(* IEC 61131-3 sources: SmartHomeNew/ (part 6) *)

(* ---- FB_Heating_Runtime_Explainability_Publisher.st ---- *)
FUNCTION_BLOCK FB_Heating_Runtime_Explainability_Publisher
VAR_INPUT
    VI_Enable : BOOL;
    VI_System_Time_MS : UDINT;
    VI_Runtime_Context : ST_Heating_Runtime_Context;
    VI_Runtime_Observation_Valid : BOOL;
    VI_Runtime_Observer_Fault : BOOL;
    VI_Runtime_Status_Code : UINT;
    VI_Runtime_Status_Text : STRING(128);
END_VAR
VAR_OUTPUT
    VO_Phase_Event : ST_Heating_Runtime_Phase_Event;
    VO_Anomaly : ST_Heating_Runtime_Anomaly;
    VO_Blackbox_Event : ST_Heating_Runtime_Blackbox_Event;
    VO_Blackbox_Timeline : ST_Heating_Runtime_Blackbox_Timeline;
    VO_Event_Buffer : ST_Heating_Runtime_Event_Buffer;
    VO_Adaptive_Intelligence : ST_Heating_Runtime_Adaptive_Intelligence;
    VO_Causality_Graph : ST_Heating_Runtime_Causality_Graph;
    VO_Integration_Bridge : ST_Heating_Runtime_Integration_Bridge;
    VO_Predictive_State : ST_Heating_Runtime_Predictive_State;
    VO_Execution_Timeline : ST_Heating_Runtime_Execution_Timeline;
    VO_Phase_Transition : ST_Heating_Runtime_Phase_Transition;
    VO_Publication_Valid : BOOL;
END_VAR
VAR
    L_Sequencing_Valid : BOOL;
    L_Ownership_Valid : BOOL;
    L_Synchronization_Valid : BOOL;
    L_Runtime_Degraded : BOOL;
    L_Status_Code : UINT;

    L_Empty_Phase_Event : ST_Heating_Runtime_Phase_Event;
    L_Empty_Anomaly : ST_Heating_Runtime_Anomaly;
    L_Empty_Blackbox_Event : ST_Heating_Runtime_Blackbox_Event;
    L_Empty_Blackbox_Timeline : ST_Heating_Runtime_Blackbox_Timeline;
    L_Empty_Event_Buffer : ST_Heating_Runtime_Event_Buffer;
    L_Empty_Adaptive_Intelligence : ST_Heating_Runtime_Adaptive_Intelligence;
    L_Empty_Causality_Graph : ST_Heating_Runtime_Causality_Graph;
    L_Empty_Integration_Bridge : ST_Heating_Runtime_Integration_Bridge;
    L_Empty_Predictive_State : ST_Heating_Runtime_Predictive_State;
    L_Empty_Execution_Timeline : ST_Heating_Runtime_Execution_Timeline;
    L_Empty_Phase_Transition : ST_Heating_Runtime_Phase_Transition;
END_VAR

// Clear complete retained output snapshots before writing current frame.
// This prevents stale array entries in timeline/event/causality structures.
VO_Phase_Event := L_Empty_Phase_Event;
VO_Anomaly := L_Empty_Anomaly;
VO_Blackbox_Event := L_Empty_Blackbox_Event;
VO_Blackbox_Timeline := L_Empty_Blackbox_Timeline;
VO_Event_Buffer := L_Empty_Event_Buffer;
VO_Adaptive_Intelligence := L_Empty_Adaptive_Intelligence;
VO_Causality_Graph := L_Empty_Causality_Graph;
VO_Integration_Bridge := L_Empty_Integration_Bridge;
VO_Predictive_State := L_Empty_Predictive_State;
VO_Execution_Timeline := L_Empty_Execution_Timeline;
VO_Phase_Transition := L_Empty_Phase_Transition;
VO_Publication_Valid := FALSE;

IF NOT VI_Enable THEN
    RETURN;
END_IF;

L_Sequencing_Valid := VI_Runtime_Context.DHW_Before_Heating_Valid AND VI_Runtime_Context.State_Publication_Before_Diagnostics_Valid;
L_Ownership_Valid := VI_Runtime_Context.OpenTherm_Ownership_Valid AND VI_Runtime_Context.Cascade_Ownership_Valid AND VI_Runtime_Context.Safety_Isolation_Valid;
L_Synchronization_Valid := VI_Runtime_Context.Output_Projection_Last_Valid;
L_Runtime_Degraded := VI_Runtime_Observer_Fault OR NOT VI_Runtime_Observation_Valid;
L_Status_Code := VI_Runtime_Status_Code;

// Phase event
VO_Phase_Event.Phase := VI_Runtime_Context.Current_Phase;
VO_Phase_Event.Event_Active := TRUE;
VO_Phase_Event.Event_Completed := VI_Runtime_Observation_Valid;
VO_Phase_Event.Event_Failed := VI_Runtime_Observer_Fault;
VO_Phase_Event.Start_Time_MS := VI_System_Time_MS;
VO_Phase_Event.End_Time_MS := VI_System_Time_MS;
VO_Phase_Event.Duration_MS := 0;
VO_Phase_Event.Ordering_Valid := VI_Runtime_Context.DHW_Before_Heating_Valid;
VO_Phase_Event.Isolation_Valid := VI_Runtime_Context.Diagnostics_Isolation_Valid;
VO_Phase_Event.Status_Code := L_Status_Code;
VO_Phase_Event.Status_Text := VI_Runtime_Status_Text;
VO_Phase_Event.Diagnostics_Visible := TRUE;
VO_Phase_Event.Explainability_Visible := TRUE;
VO_Phase_Event.Safety_Integrity_Valid := VI_Runtime_Context.Safety_Isolation_Valid;
VO_Phase_Event.OpenTherm_Ownership_Valid := VI_Runtime_Context.OpenTherm_Ownership_Valid;
VO_Phase_Event.Cascade_Ownership_Valid := VI_Runtime_Context.Cascade_Ownership_Valid;

// Phase transition snapshot
VO_Phase_Transition.Previous_Phase := VI_Runtime_Context.Current_Phase;
VO_Phase_Transition.Current_Phase := VI_Runtime_Context.Current_Phase;
VO_Phase_Transition.Next_Phase := VI_Runtime_Context.Current_Phase;
VO_Phase_Transition.Transition_Active := TRUE;
VO_Phase_Transition.Transition_Completed := VI_Runtime_Observation_Valid;
VO_Phase_Transition.Transition_Failed := VI_Runtime_Observer_Fault;
VO_Phase_Transition.Transition_Start_MS := VI_System_Time_MS;
VO_Phase_Transition.Transition_End_MS := VI_System_Time_MS;
VO_Phase_Transition.Transition_Duration_MS := 0;
VO_Phase_Transition.Sequencing_Valid := L_Sequencing_Valid;
VO_Phase_Transition.Ownership_Valid := L_Ownership_Valid;
VO_Phase_Transition.Synchronization_Valid := L_Synchronization_Valid;
VO_Phase_Transition.Status_Code := L_Status_Code;
VO_Phase_Transition.Status_Text := VI_Runtime_Status_Text;

// Anomaly
VO_Anomaly.Anomaly_Active := VI_Runtime_Observer_Fault;
VO_Anomaly.Anomaly_Acknowledged := FALSE;
VO_Anomaly.Anomaly_Cleared := NOT VI_Runtime_Observer_Fault;
VO_Anomaly.Runtime_Jitter_Detected := FALSE;
VO_Anomaly.Runtime_Latency_Detected := FALSE;
VO_Anomaly.Runtime_Degraded := L_Runtime_Degraded;
VO_Anomaly.Cascade_Degraded := NOT VI_Runtime_Context.Cascade_Ownership_Valid;
VO_Anomaly.Cascade_Boiler_Loss_Detected := FALSE;
VO_Anomaly.OpenTherm_Transport_Degraded := NOT VI_Runtime_Context.OpenTherm_Ownership_Valid;
VO_Anomaly.OpenTherm_Command_Invalid := FALSE;
VO_Anomaly.Diagnostics_Degraded := NOT VI_Runtime_Context.Diagnostics_Isolation_Valid;
VO_Anomaly.Explainability_Degraded := NOT VI_Runtime_Context.Explainability_Isolation_Valid;
VO_Anomaly.Sequencing_Invalid := NOT L_Sequencing_Valid;
VO_Anomaly.Ownership_Invalid := NOT L_Ownership_Valid;
VO_Anomaly.Synchronization_Invalid := NOT L_Synchronization_Valid;
VO_Anomaly.Severity_Level := SEL(VI_Runtime_Observer_Fault, 1, 900);
VO_Anomaly.Critical_Anomaly := VI_Runtime_Observer_Fault;
VO_Anomaly.Status_Code := L_Status_Code;
VO_Anomaly.Status_Text := VI_Runtime_Status_Text;

// Blackbox event
VO_Blackbox_Event.Event_ID := VI_System_Time_MS;
VO_Blackbox_Event.Event_Active := TRUE;
VO_Blackbox_Event.Runtime_Phase := VI_Runtime_Context.Current_Phase;
VO_Blackbox_Event.Event_Start_MS := VI_System_Time_MS;
VO_Blackbox_Event.Event_End_MS := VI_System_Time_MS;
VO_Blackbox_Event.Event_Duration_MS := 0;
VO_Blackbox_Event.Runtime_Degraded := L_Runtime_Degraded;
VO_Blackbox_Event.Runtime_Fault := VI_Runtime_Observer_Fault;
VO_Blackbox_Event.Cascade_Degraded := NOT VI_Runtime_Context.Cascade_Ownership_Valid;
VO_Blackbox_Event.Cascade_Boiler_Loss := FALSE;
VO_Blackbox_Event.OpenTherm_Degraded := NOT VI_Runtime_Context.OpenTherm_Ownership_Valid;
VO_Blackbox_Event.OpenTherm_Command_Invalid := FALSE;
VO_Blackbox_Event.Sequencing_Invalid := NOT L_Sequencing_Valid;
VO_Blackbox_Event.Ownership_Invalid := NOT L_Ownership_Valid;
VO_Blackbox_Event.Synchronization_Invalid := NOT L_Synchronization_Valid;
VO_Blackbox_Event.Root_Cause_Candidate := VI_Runtime_Observer_Fault;
VO_Blackbox_Event.Critical_Path := VI_Runtime_Observer_Fault;
VO_Blackbox_Event.Status_Code := L_Status_Code;
VO_Blackbox_Event.Status_Text := VI_Runtime_Status_Text;

// Blackbox timeline snapshot
VO_Blackbox_Timeline.Write_Index := 1;
VO_Blackbox_Timeline.Event_Count := 1;
VO_Blackbox_Timeline.Timeline_Overflow := FALSE;
VO_Blackbox_Timeline.Reconstruction_Visible := TRUE;
VO_Blackbox_Timeline.Forensic_Timeline_Visible := TRUE;
VO_Blackbox_Timeline.Root_Cause_Reconstructed := VI_Runtime_Observer_Fault;
VO_Blackbox_Timeline.Sequencing_Valid := L_Sequencing_Valid;
VO_Blackbox_Timeline.Ownership_Valid := L_Ownership_Valid;
VO_Blackbox_Timeline.Synchronization_Valid := L_Synchronization_Valid;
VO_Blackbox_Timeline.Events[1] := VO_Blackbox_Event;
VO_Blackbox_Timeline.Status_Code := L_Status_Code;
VO_Blackbox_Timeline.Status_Text := VI_Runtime_Status_Text;

// Runtime event buffer snapshot
VO_Event_Buffer.Write_Index := 1;
VO_Event_Buffer.Read_Index := 1;
VO_Event_Buffer.Event_Count := 1;
VO_Event_Buffer.Overflow := FALSE;
VO_Event_Buffer.Ordering_Integrity_Valid := L_Sequencing_Valid;
VO_Event_Buffer.Isolation_Integrity_Valid := VI_Runtime_Context.Diagnostics_Isolation_Valid;
VO_Event_Buffer.Lifecycle_Integrity_Valid := VI_Runtime_Observation_Valid;
VO_Event_Buffer.Diagnostics_Visibility_Valid := TRUE;
VO_Event_Buffer.Explainability_Visibility_Valid := TRUE;
VO_Event_Buffer.OpenTherm_Ownership_Valid := VI_Runtime_Context.OpenTherm_Ownership_Valid;
VO_Event_Buffer.Cascade_Ownership_Valid := VI_Runtime_Context.Cascade_Ownership_Valid;
VO_Event_Buffer.Safety_Ownership_Valid := VI_Runtime_Context.Safety_Isolation_Valid;
VO_Event_Buffer.Events[1] := VO_Phase_Event;
VO_Event_Buffer.Status_Code := L_Status_Code;
VO_Event_Buffer.Status_Text := VI_Runtime_Status_Text;

// Passive integration bridge
VO_Integration_Bridge.Shell_Ready := VI_Runtime_Observation_Valid;
VO_Integration_Bridge.Shell_Fault := VI_Runtime_Observer_Fault;
VO_Integration_Bridge.Shell_Contract_Valid := VI_Runtime_Observation_Valid;
VO_Integration_Bridge.Allow_DHW_Integration := VI_Runtime_Context.Allow_DHW_Phase;
VO_Integration_Bridge.Allow_Heating_Integration := VI_Runtime_Context.Allow_Heating_Phase;
VO_Integration_Bridge.Allow_Diagnostics_Integration := VI_Runtime_Context.Allow_Diagnostics_Phase;
VO_Integration_Bridge.Allow_Output_Projection_Integration := VI_Runtime_Context.Allow_Output_Projection_Phase;
VO_Integration_Bridge.Runtime_Ownership_Valid := TRUE;
VO_Integration_Bridge.Diagnostics_Ownership_Valid := VI_Runtime_Context.Diagnostics_Isolation_Valid;
VO_Integration_Bridge.Explainability_Ownership_Valid := VI_Runtime_Context.Explainability_Isolation_Valid;
VO_Integration_Bridge.OpenTherm_Ownership_Valid := VI_Runtime_Context.OpenTherm_Ownership_Valid;
VO_Integration_Bridge.Cascade_Ownership_Valid := VI_Runtime_Context.Cascade_Ownership_Valid;
VO_Integration_Bridge.Safety_Ownership_Valid := VI_Runtime_Context.Safety_Isolation_Valid;
VO_Integration_Bridge.DHW_Before_Heating_Valid := VI_Runtime_Context.DHW_Before_Heating_Valid;
VO_Integration_Bridge.Diagnostics_After_Publication_Valid := VI_Runtime_Context.State_Publication_Before_Diagnostics_Valid;
VO_Integration_Bridge.Output_Projection_Last_Valid := VI_Runtime_Context.Output_Projection_Last_Valid;
VO_Integration_Bridge.Governance_Locked := TRUE;
VO_Integration_Bridge.Runtime_Attachment_Allowed := FALSE;
VO_Integration_Bridge.Runtime_Attachment_Active := FALSE;
VO_Integration_Bridge.Integration_Status_Code := L_Status_Code;
VO_Integration_Bridge.Integration_Status_Text := VI_Runtime_Status_Text;
VO_Integration_Bridge.Diagnostics_Visible := TRUE;
VO_Integration_Bridge.Explainability_Visible := TRUE;
VO_Integration_Bridge.Current_Phase := VI_Runtime_Context.Current_Phase;
VO_Integration_Bridge.Runtime_Synchronized := L_Synchronization_Valid;

// Predictive state (passive only)
VO_Predictive_State.Predictive_Analytics_Visible := TRUE;
VO_Predictive_State.Predictive_Analytics_Degraded := L_Runtime_Degraded;
VO_Predictive_State.Predictive_Analytics_Attention := NOT VI_Runtime_Observation_Valid;
VO_Predictive_State.Runtime_Stable := NOT L_Runtime_Degraded;
VO_Predictive_State.Runtime_Stability_Score := SEL(L_Runtime_Degraded, 100, 900);
VO_Predictive_State.Runtime_Degradation_Observation := SEL(L_Runtime_Degraded, 0, 900);
VO_Predictive_State.Runtime_Failure_Observation := SEL(VI_Runtime_Observer_Fault, 0, 900);
VO_Predictive_State.Cascade_Degradation_Observation := SEL(VI_Runtime_Context.Cascade_Ownership_Valid, 900, 0);
VO_Predictive_State.Cascade_Degraded_Trend_Visible := TRUE;
VO_Predictive_State.OpenTherm_Instability_Observation := SEL(VI_Runtime_Context.OpenTherm_Ownership_Valid, 900, 0);
VO_Predictive_State.OpenTherm_Degraded_Trend_Visible := TRUE;
VO_Predictive_State.Sequencing_Observation := SEL(L_Sequencing_Valid, 900, 0);
VO_Predictive_State.Ownership_Observation := SEL(L_Ownership_Valid, 900, 0);
VO_Predictive_State.Synchronization_Observation := SEL(L_Synchronization_Valid, 900, 0);
VO_Predictive_State.Status_Code := L_Status_Code;
VO_Predictive_State.Status_Text := VI_Runtime_Status_Text;

// Execution timeline snapshot
VO_Execution_Timeline.Write_Index := 1;
VO_Execution_Timeline.Frame_Count := 1;
VO_Execution_Timeline.Timeline_Overflow := FALSE;
VO_Execution_Timeline.Sequencing_Valid := L_Sequencing_Valid;
VO_Execution_Timeline.Ownership_Valid := L_Ownership_Valid;
VO_Execution_Timeline.Synchronization_Valid := L_Synchronization_Valid;
VO_Execution_Timeline.Runtime_Jitter_Detected := FALSE;
VO_Execution_Timeline.Runtime_Latency_Detected := FALSE;
VO_Execution_Timeline.Runtime_Degraded := L_Runtime_Degraded;
VO_Execution_Timeline.Frames[1].Phase := VI_Runtime_Context.Current_Phase;
VO_Execution_Timeline.Frames[1].Frame_Started := TRUE;
VO_Execution_Timeline.Frames[1].Frame_Completed := VI_Runtime_Observation_Valid;
VO_Execution_Timeline.Frames[1].Frame_Failed := VI_Runtime_Observer_Fault;
VO_Execution_Timeline.Frames[1].Frame_Start_MS := VI_System_Time_MS;
VO_Execution_Timeline.Frames[1].Frame_End_MS := VI_System_Time_MS;
VO_Execution_Timeline.Frames[1].Frame_Duration_MS := 0;
VO_Execution_Timeline.Frames[1].Sequencing_Valid := L_Sequencing_Valid;
VO_Execution_Timeline.Frames[1].Ownership_Valid := L_Ownership_Valid;
VO_Execution_Timeline.Frames[1].Synchronization_Valid := L_Synchronization_Valid;
VO_Execution_Timeline.Frames[1].Runtime_Jitter_Detected := FALSE;
VO_Execution_Timeline.Frames[1].Runtime_Latency_Detected := FALSE;
VO_Execution_Timeline.Frames[1].Runtime_Degraded := L_Runtime_Degraded;
VO_Execution_Timeline.Frames[1].Status_Code := L_Status_Code;
VO_Execution_Timeline.Frames[1].Status_Text := VI_Runtime_Status_Text;
VO_Execution_Timeline.Status_Code := L_Status_Code;
VO_Execution_Timeline.Status_Text := VI_Runtime_Status_Text;

// Adaptive intelligence (passive only)
VO_Adaptive_Intelligence.Adaptive_Analytics_Visible := TRUE;
VO_Adaptive_Intelligence.Adaptive_Analytics_Degraded := L_Runtime_Degraded;
VO_Adaptive_Intelligence.Adaptive_Analytics_Attention := NOT VI_Runtime_Observation_Valid;
VO_Adaptive_Intelligence.Supervision_Confidence_Observation := SEL(L_Runtime_Degraded, 100, 900);
VO_Adaptive_Intelligence.Confidence_Degradation_Visible := L_Runtime_Degraded;
VO_Adaptive_Intelligence.Adaptive_Runtime_Observation := 1;
VO_Adaptive_Intelligence.Adaptive_Runtime_Stability_Observation := SEL(L_Runtime_Degraded, 100, 900);
VO_Adaptive_Intelligence.Runtime_Anomaly_Observation_Weight := 1;
VO_Adaptive_Intelligence.Cascade_Anomaly_Observation_Weight := 1;
VO_Adaptive_Intelligence.OpenTherm_Anomaly_Observation_Weight := 1;
VO_Adaptive_Intelligence.Diagnostics_Anomaly_Observation_Weight := 1;
VO_Adaptive_Intelligence.Predictive_Correlation_Observation := 1;
VO_Adaptive_Intelligence.Predictive_Correlation_Visible := TRUE;
VO_Adaptive_Intelligence.Sequencing_Confidence_Observation := SEL(L_Sequencing_Valid, 100, 900);
VO_Adaptive_Intelligence.Ownership_Confidence_Observation := SEL(L_Ownership_Valid, 100, 900);
VO_Adaptive_Intelligence.Synchronization_Confidence_Observation := SEL(L_Synchronization_Valid, 100, 900);
VO_Adaptive_Intelligence.Status_Code := L_Status_Code;
VO_Adaptive_Intelligence.Status_Text := VI_Runtime_Status_Text;

// Minimal causality graph snapshot
VO_Causality_Graph.Node_Count := 1;
VO_Causality_Graph.Edge_Count := 1;
VO_Causality_Graph.Graph_Active := TRUE;
VO_Causality_Graph.Graph_Degraded := L_Runtime_Degraded;
VO_Causality_Graph.Graph_Critical := VI_Runtime_Observer_Fault;
VO_Causality_Graph.Sequencing_Valid := L_Sequencing_Valid;
VO_Causality_Graph.Ownership_Valid := L_Ownership_Valid;
VO_Causality_Graph.Synchronization_Valid := L_Synchronization_Valid;
VO_Causality_Graph.Nodes[1].Node_ID := 1;
VO_Causality_Graph.Nodes[1].Node_Active := TRUE;
VO_Causality_Graph.Nodes[1].Runtime_Degraded := L_Runtime_Degraded;
VO_Causality_Graph.Nodes[1].Runtime_Fault := VI_Runtime_Observer_Fault;
VO_Causality_Graph.Nodes[1].Cascade_Degraded := NOT VI_Runtime_Context.Cascade_Ownership_Valid;
VO_Causality_Graph.Nodes[1].OpenTherm_Degraded := NOT VI_Runtime_Context.OpenTherm_Ownership_Valid;
VO_Causality_Graph.Nodes[1].Diagnostics_Degraded := NOT VI_Runtime_Context.Diagnostics_Isolation_Valid;
VO_Causality_Graph.Nodes[1].Explainability_Degraded := NOT VI_Runtime_Context.Explainability_Isolation_Valid;
VO_Causality_Graph.Nodes[1].Sequencing_Invalid := NOT L_Sequencing_Valid;
VO_Causality_Graph.Nodes[1].Ownership_Invalid := NOT L_Ownership_Valid;
VO_Causality_Graph.Nodes[1].Synchronization_Invalid := NOT L_Synchronization_Valid;
VO_Causality_Graph.Nodes[1].Severity_Level := SEL(VI_Runtime_Observer_Fault, 1, 900);
VO_Causality_Graph.Nodes[1].Root_Cause_Candidate := VI_Runtime_Observer_Fault;
VO_Causality_Graph.Nodes[1].Status_Code := L_Status_Code;
VO_Causality_Graph.Nodes[1].Status_Text := VI_Runtime_Status_Text;
VO_Causality_Graph.Edges[1].Source_Node_ID := 1;
VO_Causality_Graph.Edges[1].Target_Node_ID := 1;
VO_Causality_Graph.Edges[1].Edge_Active := TRUE;
VO_Causality_Graph.Edges[1].Propagation_Detected := L_Runtime_Degraded;
VO_Causality_Graph.Edges[1].Runtime_Propagation := L_Runtime_Degraded;
VO_Causality_Graph.Edges[1].Cascade_Propagation := NOT VI_Runtime_Context.Cascade_Ownership_Valid;
VO_Causality_Graph.Edges[1].OpenTherm_Propagation := NOT VI_Runtime_Context.OpenTherm_Ownership_Valid;
VO_Causality_Graph.Edges[1].Diagnostics_Propagation := NOT VI_Runtime_Context.Diagnostics_Isolation_Valid;
VO_Causality_Graph.Edges[1].Sequencing_Propagation := NOT L_Sequencing_Valid;
VO_Causality_Graph.Edges[1].Ownership_Propagation := NOT L_Ownership_Valid;
VO_Causality_Graph.Edges[1].Synchronization_Propagation := NOT L_Synchronization_Valid;
VO_Causality_Graph.Status_Code := L_Status_Code;
VO_Causality_Graph.Status_Text := VI_Runtime_Status_Text;

VO_Publication_Valid := TRUE;

END_FUNCTION_BLOCK
// >>> BULK_SYNC_ANCHOR: FB_Heating_Runtime_Explainability_Publisher <<<

(* ---- FB_Heating_Runtime_Fault_Replay_Analyzer.st ---- *)
// ==============================================================================
// Heating runtime fault replay analyzer
// Read-only runtime forensic replay layer.
// ==============================================================================
FUNCTION_BLOCK FB_Heating_Runtime_Fault_Replay_Analyzer
VAR_INPUT
    VI_Enable : BOOL;
    VI_Event : ST_Heating_Runtime_Blackbox_Event;
END_VAR
VAR_OUTPUT
    VO_Replay_Active : BOOL;
    VO_Root_Cause_Reconstructed : BOOL;

    VO_Status_Code : UINT;
    VO_Status_Text : STRING(128);
END_VAR

VO_Replay_Active := FALSE;
VO_Root_Cause_Reconstructed := FALSE;

VO_Status_Code := 0;
VO_Status_Text := 'Heating runtime replay analyzer disabled';

IF NOT VI_Enable THEN
    RETURN;
END_IF;

VO_Replay_Active := VI_Event.Event_Active;

VO_Root_Cause_Reconstructed :=
    VI_Event.Root_Cause_Candidate OR
    VI_Event.Critical_Path OR
    VI_Event.Sequencing_Invalid OR
    VI_Event.Ownership_Invalid OR
    VI_Event.Synchronization_Invalid;

IF VO_Root_Cause_Reconstructed THEN
    VO_Status_Code := 900;
    VO_Status_Text := 'Heating runtime fault replay reconstructed';
ELSE
    VO_Status_Code := 1;
    VO_Status_Text := 'Heating runtime replay nominal';
END_IF;

END_FUNCTION_BLOCK
// >>> BULK_SYNC_ANCHOR: FB_Heating_Runtime_Fault_Replay_Analyzer <<<

(* ---- FB_Heating_Runtime_Integration_Bridge_Manager.st ---- *)
// ==============================================================================
// Heating runtime integration bridge manager
// Read-only orchestration integration layer.
// DOES NOT own runtime.
// DOES NOT own heating logic.
// DOES NOT own diagnostics.
// DOES NOT own OpenTherm transport.
// DOES NOT connect orchestration to live runtime yet.
// ==============================================================================
FUNCTION_BLOCK FB_Heating_Runtime_Integration_Bridge_Manager
VAR_INPUT
    VI_Enable : BOOL;
    VI_Runtime_Context : ST_Heating_Runtime_Context;
    VI_Contract_Valid : BOOL;
END_VAR
VAR_OUTPUT
    VO_Bridge : ST_Heating_Runtime_Integration_Bridge;

    VO_Bridge_Ready : BOOL;
    VO_Bridge_Fault : BOOL;
    VO_Bridge_Status_Code : UINT;
    VO_Bridge_Status_Text : STRING(128);
END_VAR

// ======================================================
// DEFAULTS
// ======================================================
VO_Bridge.Shell_Ready := FALSE;
VO_Bridge.Shell_Fault := FALSE;
VO_Bridge.Shell_Contract_Valid := FALSE;

VO_Bridge.Allow_DHW_Integration := FALSE;
VO_Bridge.Allow_Heating_Integration := FALSE;
VO_Bridge.Allow_Diagnostics_Integration := FALSE;
VO_Bridge.Allow_Output_Projection_Integration := FALSE;

VO_Bridge.Runtime_Ownership_Valid := TRUE;
VO_Bridge.Diagnostics_Ownership_Valid := TRUE;
VO_Bridge.Explainability_Ownership_Valid := TRUE;
VO_Bridge.OpenTherm_Ownership_Valid := TRUE;
VO_Bridge.Cascade_Ownership_Valid := TRUE;
VO_Bridge.Safety_Ownership_Valid := TRUE;

VO_Bridge.DHW_Before_Heating_Valid := TRUE;
VO_Bridge.Diagnostics_After_Publication_Valid := TRUE;
VO_Bridge.Output_Projection_Last_Valid := TRUE;

// ======================================================
// GOVERNANCE LOCK
// Migration is NEVER auto-enabled by supervision.
// ======================================================
VO_Bridge.Runtime_Migration_Allowed := FALSE;
VO_Bridge.Runtime_Migration_Active := FALSE;
VO_Bridge.Runtime_Migration_Failed := FALSE;

VO_Bridge.Integration_Status_Code := 0;
VO_Bridge.Integration_Status_Text := 'Heating runtime bridge disabled';

VO_Bridge.Diagnostics_Visible := TRUE;
VO_Bridge.Explainability_Visible := TRUE;

VO_Bridge.Current_Phase := E_Heating_Runtime_Phase.HRP_DISABLED;
VO_Bridge.Runtime_Synchronized := FALSE;

VO_Bridge_Ready := FALSE;
VO_Bridge_Fault := FALSE;
VO_Bridge_Status_Code := 0;
VO_Bridge_Status_Text := 'Heating runtime bridge disabled';

IF NOT VI_Enable THEN
    RETURN;
END_IF;

// ======================================================
// SHELL STATE
// ======================================================
VO_Bridge.Shell_Ready := VI_Runtime_Context.Runtime_Ready;
VO_Bridge.Shell_Fault := VI_Runtime_Context.Runtime_Fault;
VO_Bridge.Shell_Contract_Valid := VI_Contract_Valid;

// ======================================================
// OWNERSHIP INTEGRITY
// ======================================================
VO_Bridge.Runtime_Ownership_Valid := TRUE;

VO_Bridge.Diagnostics_Ownership_Valid :=
    VI_Runtime_Context.Diagnostics_Isolation_Valid;

VO_Bridge.Explainability_Ownership_Valid :=
    VI_Runtime_Context.Explainability_Isolation_Valid;

VO_Bridge.OpenTherm_Ownership_Valid :=
    VI_Runtime_Context.OpenTherm_Ownership_Valid;

VO_Bridge.Cascade_Ownership_Valid :=
    VI_Runtime_Context.Cascade_Ownership_Valid;

VO_Bridge.Safety_Ownership_Valid :=
    VI_Runtime_Context.Safety_Isolation_Valid;

// ======================================================
// SEQUENCING INTEGRITY
// ======================================================
VO_Bridge.DHW_Before_Heating_Valid :=
    VI_Runtime_Context.DHW_Before_Heating_Valid;

VO_Bridge.Diagnostics_After_Publication_Valid :=
    VI_Runtime_Context.State_Publication_Before_Diagnostics_Valid;

VO_Bridge.Output_Projection_Last_Valid :=
    VI_Runtime_Context.Output_Projection_Last_Valid;

// ======================================================
// OBSERVATION-ONLY INTEGRATION READINESS
// ======================================================
VO_Bridge.Allow_DHW_Integration :=
    VO_Bridge.DHW_Before_Heating_Valid;

VO_Bridge.Allow_Heating_Integration :=
    VO_Bridge.Runtime_Ownership_Valid AND
    VO_Bridge.Cascade_Ownership_Valid;

VO_Bridge.Allow_Diagnostics_Integration :=
    VO_Bridge.Diagnostics_Ownership_Valid AND
    VO_Bridge.Explainability_Ownership_Valid;

VO_Bridge.Allow_Output_Projection_Integration :=
    VO_Bridge.Output_Projection_Last_Valid;

// ======================================================
// GOVERNANCE POLICY
// Runtime migration is NOT automatically allowed.
// Future migration requires explicit external governance.
// ======================================================
VO_Bridge.Runtime_Migration_Allowed := FALSE;
VO_Bridge.Runtime_Migration_Active := FALSE;
VO_Bridge.Runtime_Migration_Failed := FALSE;

// ======================================================
// PHASE SYNCHRONIZATION
// ======================================================
VO_Bridge.Current_Phase := VI_Runtime_Context.Current_Phase;
VO_Bridge.Runtime_Synchronized := VI_Contract_Valid;

// ======================================================
// STATUS
// ======================================================
IF NOT VI_Contract_Valid THEN
    VO_Bridge.Integration_Status_Code := 100;
    VO_Bridge.Integration_Status_Text := 'Heating runtime contract invalid';

ELSIF VI_Runtime_Context.Runtime_Fault THEN
    VO_Bridge.Integration_Status_Code := 200;
    VO_Bridge.Integration_Status_Text := 'Heating runtime fault active';

ELSIF NOT VO_Bridge.Allow_Heating_Integration THEN
    VO_Bridge.Integration_Status_Code := 300;
    VO_Bridge.Integration_Status_Text := 'Heating observation integration blocked';

ELSE
    VO_Bridge.Integration_Status_Code := 1;
    VO_Bridge.Integration_Status_Text := 'Heating observation bridge ready';
END_IF;

// ======================================================
// OUTPUT STATUS
// ======================================================
VO_Bridge_Ready :=
    VO_Bridge.Allow_Heating_Integration;

VO_Bridge_Fault :=
    NOT VI_Contract_Valid OR
    VI_Runtime_Context.Runtime_Fault;

VO_Bridge_Status_Code :=
    VO_Bridge.Integration_Status_Code;

VO_Bridge_Status_Text :=
    VO_Bridge.Integration_Status_Text;

END_FUNCTION_BLOCK
// >>> BULK_SYNC_ANCHOR: FB_Heating_Runtime_Integration_Bridge_Manager <<<

(* ---- FB_Heating_Runtime_Intelligence_Consistency_Analyzer.st ---- *)
// ==============================================================================
// Heating runtime intelligence consistency analyzer
// Read-only meta-supervision consistency layer.
// ==============================================================================
FUNCTION_BLOCK FB_Heating_Runtime_Intelligence_Consistency_Analyzer
VAR_INPUT
    VI_Enable : BOOL;
    VI_Integrity_Valid : BOOL;
    VI_Drift_Detected : BOOL;
    VI_Decay_Detected : BOOL;
END_VAR
VAR_OUTPUT
    VO_Consistency_Valid : BOOL;
    VO_Consistency_Score : UINT;

    VO_Status_Code : UINT;
    VO_Status_Text : STRING(128);
END_VAR

VO_Consistency_Valid := FALSE;
VO_Consistency_Score := 0;

VO_Status_Code := 0;
VO_Status_Text := 'Heating intelligence consistency analyzer disabled';

IF NOT VI_Enable THEN
    RETURN;
END_IF;

VO_Consistency_Valid :=
    VI_Integrity_Valid AND
    NOT VI_Drift_Detected AND
    NOT VI_Decay_Detected;

IF VO_Consistency_Valid THEN
    VO_Consistency_Score := 95;

    VO_Status_Code := 1;
    VO_Status_Text := 'Heating intelligence consistency nominal';

ELSIF VI_Integrity_Valid THEN
    VO_Consistency_Score := 60;

    VO_Status_Code := 200;
    VO_Status_Text := 'Heating intelligence consistency degraded';

ELSE
    VO_Consistency_Score := 10;

    VO_Status_Code := 900;
    VO_Status_Text := 'Heating intelligence consistency invalid';
END_IF;

END_FUNCTION_BLOCK
// >>> BULK_SYNC_ANCHOR: FB_Heating_Runtime_Intelligence_Consistency_Analyzer <<<

(* ---- FB_Heating_Runtime_Latency_Validator.st ---- *)
// ==============================================================================
// Heating runtime latency validator
// Read-only deterministic execution latency validator.
// ==============================================================================
FUNCTION_BLOCK FB_Heating_Runtime_Latency_Validator
VAR_INPUT
    VI_Enable : BOOL;
    VI_Frame_Duration_MS : UDINT;
END_VAR
VAR_OUTPUT
    VO_Latency_Detected : BOOL;
    VO_Runtime_Degraded : BOOL;

    VO_Status_Code : UINT;
    VO_Status_Text : STRING(128);
END_VAR

VO_Latency_Detected := FALSE;
VO_Runtime_Degraded := FALSE;

VO_Status_Code := 0;
VO_Status_Text := 'Heating runtime latency validator disabled';

IF NOT VI_Enable THEN
    RETURN;
END_IF;

IF VI_Frame_Duration_MS > 1000 THEN
    VO_Latency_Detected := TRUE;
    VO_Runtime_Degraded := TRUE;

    VO_Status_Code := 900;
    VO_Status_Text := 'Heating runtime latency critical';

ELSIF VI_Frame_Duration_MS > 500 THEN
    VO_Latency_Detected := TRUE;

    VO_Status_Code := 200;
    VO_Status_Text := 'Heating runtime latency degraded';

ELSE
    VO_Status_Code := 1;
    VO_Status_Text := 'Heating runtime latency nominal';
END_IF;

END_FUNCTION_BLOCK
// >>> BULK_SYNC_ANCHOR: FB_Heating_Runtime_Latency_Validator <<<

(* ---- FB_Heating_Runtime_Meta_Supervision_Publisher.st ---- *)
FUNCTION_BLOCK FB_Heating_Runtime_Meta_Supervision_Publisher
VAR_INPUT
    VI_Enable : BOOL;
    VI_Runtime_Observation_Valid : BOOL;
    VI_Runtime_Observer_Ready : BOOL;
    VI_Runtime_Observer_Fault : BOOL;
    VI_Runtime_Status_Code : UINT;
    VI_Runtime_Status_Text : STRING(128);
END_VAR
VAR_OUTPUT
    VO_Meta : ST_Heating_Runtime_Meta_Supervision;
    VO_Publication_Valid : BOOL;
END_VAR

VO_Meta.Meta_Analytics_Visible := FALSE;
VO_Meta.Meta_Analytics_Degraded := FALSE;
VO_Meta.Meta_Analytics_Attention := FALSE;

VO_Meta.Supervision_Integrity_Visible := FALSE;
VO_Meta.Supervision_Integrity_Observation := 0;

VO_Meta.Adaptive_Drift_Visible := FALSE;
VO_Meta.Adaptive_Drift_Observation := 0;

VO_Meta.Confidence_Degradation_Visible := FALSE;
VO_Meta.Confidence_Degradation_Observation := 0;

VO_Meta.Analytics_Consistency_Visible := FALSE;
VO_Meta.Analytics_Consistency_Observation := 0;

VO_Meta.Sequencing_Meta_Observation := FALSE;
VO_Meta.Ownership_Meta_Observation := FALSE;
VO_Meta.Synchronization_Meta_Observation := FALSE;

VO_Meta.Status_Code := 0;
VO_Meta.Status_Text := 'Heating runtime meta supervision inactive';

VO_Publication_Valid := FALSE;

IF NOT VI_Enable THEN
    RETURN;
END_IF;

VO_Meta.Meta_Analytics_Visible := TRUE;
VO_Meta.Supervision_Integrity_Visible := TRUE;
VO_Meta.Adaptive_Drift_Visible := TRUE;
VO_Meta.Confidence_Degradation_Visible := TRUE;
VO_Meta.Analytics_Consistency_Visible := TRUE;

VO_Meta.Sequencing_Meta_Observation := VI_Runtime_Observation_Valid;
VO_Meta.Ownership_Meta_Observation := VI_Runtime_Observer_Ready;
VO_Meta.Synchronization_Meta_Observation := NOT VI_Runtime_Observer_Fault;

IF VI_Runtime_Observer_Fault THEN
    VO_Meta.Meta_Analytics_Degraded := TRUE;
    VO_Meta.Meta_Analytics_Attention := TRUE;
    VO_Meta.Supervision_Integrity_Observation := 900;
ELSIF NOT VI_Runtime_Observation_Valid THEN
    VO_Meta.Meta_Analytics_Attention := TRUE;
    VO_Meta.Supervision_Integrity_Observation := 200;
ELSE
    VO_Meta.Supervision_Integrity_Observation := 1;
END_IF;

VO_Meta.Status_Code := VI_Runtime_Status_Code;
VO_Meta.Status_Text := VI_Runtime_Status_Text;

VO_Publication_Valid := TRUE;

END_FUNCTION_BLOCK
// >>> BULK_SYNC_ANCHOR: FB_Heating_Runtime_Meta_Supervision_Publisher <<<

(* ---- FB_Heating_Runtime_Observability.st ---- *)
// ==============================================================================
// Heating runtime observability layer
//
// Projection/publication layer only.
//
// IMPORTANT:
// - does NOT own outputs;
// - does NOT control pumps/valves;
// - does NOT modify demand;
// - does NOT participate in runtime authority.
//
// Responsibility:
// - allocation snapshot publication;
// - policy diagnostics projection;
// - freeze/DHW bypass visibility;
// - runtime explainability;
// - bounded policy bridge visibility.
// ==============================================================================
FUNCTION_BLOCK FB_Heating_Runtime_Observability
VAR_INPUT
    VI_Policy_Active : BOOL;
    VI_Freeze_Bypass_Active : BOOL;
    VI_DHW_Bypass_Active : BOOL;

    VI_Budget_Max : REAL;
    VI_Budget_Used : REAL;

    VI_Requested : ARRAY[1..GVL_CONSTANTS.C_MAX_MANIFOLDS] OF BOOL;
    VI_Allowed : ARRAY[1..GVL_CONSTANTS.C_MAX_MANIFOLDS] OF BOOL;
    VI_Filtered : ARRAY[1..GVL_CONSTANTS.C_MAX_MANIFOLDS] OF BOOL;

    VI_Block_Reason : ARRAY[1..GVL_CONSTANTS.C_MAX_MANIFOLDS] OF E_Heating_Allocation_Block_Reason;
    VI_Effective_Priority : ARRAY[1..GVL_CONSTANTS.C_MAX_MANIFOLDS] OF INT;
END_VAR
VAR
    L_i : INT;
    L_Policy_Target_Adjustment : REAL;
    L_Policy_Priority_Multiplier : REAL;
END_VAR

GVL_STATE.G_Allocation_Policy_Active := VI_Policy_Active;
GVL_STATE.G_Allocation_Freeze_Bypass_Active := VI_Freeze_Bypass_Active;
GVL_STATE.G_Allocation_DHW_Bypass_Active := VI_DHW_Bypass_Active;

GVL_STATE.G_Allocation_Budget_Max := VI_Budget_Max;
GVL_STATE.G_Allocation_Budget_Used := VI_Budget_Used;

FOR L_i := 1 TO GVL_CONSTANTS.C_MAX_MANIFOLDS DO
    GVL_STATE.G_Allocation_Requested[L_i] := VI_Requested[L_i];
    GVL_STATE.G_Allocation_Allowed[L_i] := VI_Allowed[L_i];
    GVL_STATE.G_Allocation_Filtered[L_i] := VI_Filtered[L_i];

    GVL_STATE.G_Allocation_Block_Reason[L_i] := VI_Block_Reason[L_i];
    GVL_STATE.G_Allocation_Effective_Priority[L_i] := VI_Effective_Priority[L_i];
END_FOR;

// Bounded policy bridge visibility.
// Mirrors the same clamp used by FB_Heating_System_Manager.
L_Policy_Target_Adjustment := GVL_HEATING_POLICY.G_Policy_Target_Adjustment;
IF L_Policy_Target_Adjustment > REAL#5.0 THEN
    L_Policy_Target_Adjustment := REAL#5.0;
ELSIF L_Policy_Target_Adjustment < REAL#-3.0 THEN
    L_Policy_Target_Adjustment := REAL#-3.0;
END_IF;

L_Policy_Priority_Multiplier := GVL_HEATING_POLICY.G_Policy_Priority_Multiplier;
IF L_Policy_Priority_Multiplier < REAL#0.3 THEN
    L_Policy_Priority_Multiplier := REAL#0.3;
ELSIF L_Policy_Priority_Multiplier > REAL#1.0 THEN
    L_Policy_Priority_Multiplier := REAL#1.0;
END_IF;

GVL_STATE.G_Policy_Target_Adjustment_Applied := L_Policy_Target_Adjustment;
GVL_STATE.G_Policy_Target_Adjustment_Active := ABS(L_Policy_Target_Adjustment) > REAL#0.001;
GVL_STATE.G_Policy_Priority_Multiplier_Applied := L_Policy_Priority_Multiplier;

END_FUNCTION_BLOCK
// >>> BULK_SYNC_ANCHOR: FB_Heating_Runtime_Observability <<<

(* ---- FB_Heating_Runtime_Observer.st ---- *)
// ==============================================================================
// Heating runtime observer
// Minimal observer-only runtime attachment.
// Read-only.
// Governance-locked.
// Finalized-state observation only.
// ==============================================================================
FUNCTION_BLOCK FB_Heating_Runtime_Observer
VAR_INPUT
    VI_Enable : BOOL;
    VI_Runtime_Context : ST_Heating_Runtime_Context;
    VI_Diagnostics_Valid : BOOL;
END_VAR
VAR_OUTPUT
    VO_Observation : ST_Heating_Runtime_Observation;

    VO_Observer_Ready : BOOL;
    VO_Observer_Fault : BOOL;
    VO_Status_Code : UINT;
    VO_Status_Text : STRING(128);
END_VAR

// ======================================================
// DEFAULTS
// ======================================================
VO_Observation.Runtime_Visible := FALSE;
VO_Observation.Diagnostics_Visible := FALSE;
VO_Observation.OT_Visible := FALSE;
VO_Observation.Cascade_Visible := FALSE;

VO_Observation.Runtime_Ready := FALSE;
VO_Observation.Runtime_Fault := FALSE;
VO_Observation.Diagnostics_Valid := FALSE;

VO_Observation.Current_Phase := E_Heating_Runtime_Phase.HRP_DISABLED;

VO_Observation.Sequencing_Visible := FALSE;
VO_Observation.Ownership_Visible := FALSE;
VO_Observation.Synchronization_Visible := FALSE;

VO_Observation.Status_Code := 0;
VO_Observation.Status_Text := 'Heating runtime observer disabled';

VO_Observer_Ready := FALSE;
VO_Observer_Fault := FALSE;
VO_Status_Code := 0;
VO_Status_Text := 'Heating runtime observer disabled';

IF NOT VI_Enable THEN
    RETURN;
END_IF;

// ======================================================
// FINALIZED-STATE OBSERVATION ONLY
// ======================================================
VO_Observation.Runtime_Visible := TRUE;
VO_Observation.Diagnostics_Visible := TRUE;
VO_Observation.OT_Visible := TRUE;
VO_Observation.Cascade_Visible := TRUE;

VO_Observation.Runtime_Ready :=
    VI_Runtime_Context.Runtime_Ready;

VO_Observation.Runtime_Fault :=
    VI_Runtime_Context.Runtime_Fault;

VO_Observation.Diagnostics_Valid :=
    VI_Diagnostics_Valid;

VO_Observation.Current_Phase :=
    VI_Runtime_Context.Current_Phase;

VO_Observation.Sequencing_Visible :=
    VI_Runtime_Context.DHW_Before_Heating_Valid;

VO_Observation.Ownership_Visible :=
    VI_Runtime_Context.Cascade_Ownership_Valid AND
    VI_Runtime_Context.OpenTherm_Ownership_Valid;

VO_Observation.Synchronization_Visible :=
    VI_Runtime_Context.State_Publication_Before_Diagnostics_Valid;

// ======================================================
// STATUS
// ======================================================
IF VI_Runtime_Context.Runtime_Fault THEN
    VO_Observation.Status_Code := 900;
    VO_Observation.Status_Text := 'Heating runtime observer detected runtime fault';

ELSIF NOT VI_Diagnostics_Valid THEN
    VO_Observation.Status_Code := 200;
    VO_Observation.Status_Text := 'Heating runtime diagnostics publication invalid';

ELSE
    VO_Observation.Status_Code := 1;
    VO_Observation.Status_Text := 'Heating runtime observer nominal';
END_IF;

VO_Observer_Ready := TRUE;
VO_Observer_Fault := FALSE;

VO_Status_Code := VO_Observation.Status_Code;
VO_Status_Text := VO_Observation.Status_Text;

END_FUNCTION_BLOCK
// >>> BULK_SYNC_ANCHOR: FB_Heating_Runtime_Observer <<<

(* ---- FB_Heating_Runtime_Observer_Authorization.st ---- *)
// ==============================================================================
// Heating runtime observer authorization
// Governed passive-bootstrap authorization only.
// Read-only.
// Deterministic.
// ==============================================================================
FUNCTION_BLOCK FB_Heating_Runtime_Observer_Authorization
VAR_INPUT
    VI_Enable_Request : BOOL;

    VI_Bootstrap_Mode : BOOL;
    VI_Passive_Mode : BOOL;
    VI_ReadOnly_Mode : BOOL;

    VI_Governance_Locked : BOOL;
    VI_Runtime_Authority_Disabled : BOOL;
    VI_Writable_Exports_Disabled : BOOL;
END_VAR
VAR_OUTPUT
    VO_Enable_Authorized : BOOL;
    VO_Enable_Effective : BOOL;

    VO_Authorization_Valid : BOOL;

    VO_Deny_Reason : E_Runtime_Observer_Deny_Reason;
    VO_Deny_Text : STRING(128);

    VO_Status_Code : UINT;
    VO_Status_Text : STRING(128);
END_VAR

// ======================================================
// DEFAULTS
// ======================================================
VO_Enable_Authorized := FALSE;
VO_Enable_Effective := FALSE;
VO_Authorization_Valid := FALSE;

VO_Deny_Reason := E_Runtime_Observer_Deny_Reason.RODR_NONE;
VO_Deny_Text := 'No deny reason';

VO_Status_Code := 0;
VO_Status_Text := 'Heating runtime observer authorization inactive';

// ======================================================
// REQUEST VALIDATION
// ======================================================
IF NOT VI_Enable_Request THEN
    VO_Deny_Reason := E_Runtime_Observer_Deny_Reason.RODR_NO_ENABLE_REQUEST;
    VO_Deny_Text := 'Observer enable request is not active';
    RETURN;
END_IF;

// ======================================================
// GOVERNANCE VALIDATION
// ======================================================
IF NOT VI_Bootstrap_Mode THEN
    VO_Deny_Reason := E_Runtime_Observer_Deny_Reason.RODR_BOOTSTRAP_DISABLED;
    VO_Deny_Text := 'Bootstrap mode required for observer authorization';
    VO_Status_Code := 100;
    VO_Status_Text := 'Bootstrap mode required for observer authorization';
    RETURN;
END_IF;

IF NOT VI_Passive_Mode THEN
    VO_Deny_Reason := E_Runtime_Observer_Deny_Reason.RODR_PASSIVE_MODE_DISABLED;
    VO_Deny_Text := 'Passive mode required for observer authorization';
    VO_Status_Code := 110;
    VO_Status_Text := 'Passive mode required for observer authorization';
    RETURN;
END_IF;

IF NOT VI_ReadOnly_Mode THEN
    VO_Deny_Reason := E_Runtime_Observer_Deny_Reason.RODR_READONLY_MODE_DISABLED;
    VO_Deny_Text := 'Read-only mode required for observer authorization';
    VO_Status_Code := 120;
    VO_Status_Text := 'Read-only mode required for observer authorization';
    RETURN;
END_IF;

IF NOT VI_Governance_Locked THEN
    VO_Deny_Reason := E_Runtime_Observer_Deny_Reason.RODR_GOVERNANCE_UNLOCKED;
    VO_Deny_Text := 'Governance lock required for observer authorization';
    VO_Status_Code := 130;
    VO_Status_Text := 'Governance lock required for observer authorization';
    RETURN;
END_IF;

IF NOT VI_Runtime_Authority_Disabled THEN
    VO_Deny_Reason := E_Runtime_Observer_Deny_Reason.RODR_RUNTIME_AUTHORITY_ENABLED;
    VO_Deny_Text := 'Runtime authority isolation required';
    VO_Status_Code := 140;
    VO_Status_Text := 'Runtime authority isolation required';
    RETURN;
END_IF;

IF NOT VI_Writable_Exports_Disabled THEN
    VO_Deny_Reason := E_Runtime_Observer_Deny_Reason.RODR_WRITABLE_EXPORTS_ENABLED;
    VO_Deny_Text := 'Writable exports must remain disabled';
    VO_Status_Code := 150;
    VO_Status_Text := 'Writable exports must remain disabled';
    RETURN;
END_IF;

// ======================================================
// AUTHORIZED PASSIVE BOOTSTRAP ACTIVATION
// ======================================================
VO_Enable_Authorized := TRUE;
VO_Enable_Effective := TRUE;
VO_Authorization_Valid := TRUE;

VO_Deny_Reason := E_Runtime_Observer_Deny_Reason.RODR_NONE;
VO_Deny_Text := 'No deny reason';

VO_Status_Code := 1;
VO_Status_Text := 'Heating runtime observer authorization granted';

END_FUNCTION_BLOCK
// >>> BULK_SYNC_ANCHOR: FB_Heating_Runtime_Observer_Authorization <<<

(* ---- FB_Heating_Runtime_Orchestration_Shell.st ---- *)
// ==============================================================================
// Heating runtime orchestration shell
// Prepared integration boundary for future controlled extraction.
// DOES NOT own heating logic.
// DOES NOT own diagnostics.
// DOES NOT own OpenTherm transport.
// DOES NOT own safety.
// NOT connected to live runtime yet.
// ==============================================================================
FUNCTION_BLOCK FB_Heating_Runtime_Orchestration_Shell
VAR_INPUT
    VI_Enable : BOOL;
    VI_System_Time_MS : UDINT;
END_VAR
VAR_OUTPUT
    VO_Runtime_Context : ST_Heating_Runtime_Context;
    VO_Runtime_Event_Buffer : ST_Heating_Runtime_Event_Buffer;

    VO_Contract_Valid : BOOL;
    VO_Runtime_Ready : BOOL;
    VO_Runtime_Fault : BOOL;
    VO_Status_Code : UINT;
    VO_Status_Text : STRING(128);
END_VAR
VAR
    fbCoordinator : FB_Heating_Runtime_Coordinator;
    fbValidator : FB_Heating_Runtime_Contract_Validator;
    fbEventManager : FB_Heating_Runtime_Event_Manager;

    L_Event : ST_Heating_Runtime_Phase_Event;
    L_Event_Stored : BOOL;
    L_Buffer_Overflow : BOOL;
    L_Event_Manager_Ready : BOOL;
    L_Event_Manager_Code : UINT;
    L_Event_Manager_Text : STRING(128);
END_VAR

// ======================================================
// DEFAULTS
// ======================================================
VO_Contract_Valid := FALSE;
VO_Runtime_Ready := FALSE;
VO_Runtime_Fault := FALSE;
VO_Status_Code := 0;
VO_Status_Text := 'Heating runtime orchestration shell disabled';

IF NOT VI_Enable THEN
    RETURN;
END_IF;

// ======================================================
// COORDINATION CONTEXT
// ======================================================
fbCoordinator(
    VI_Enable := VI_Enable,
    VO_Runtime_Context => VO_Runtime_Context
);

// ======================================================
// CONTRACT VALIDATION
// ======================================================
fbValidator(
    VI_Context := VO_Runtime_Context,
    VO_Contract_Valid => VO_Contract_Valid
);

// ======================================================
// PHASE EVENT PROJECTION
// ======================================================
L_Event.Phase := VO_Runtime_Context.Current_Phase;
L_Event.Event_Active := VI_Enable;
L_Event.Event_Completed := VO_Runtime_Context.Runtime_Ready;
L_Event.Event_Failed := VO_Runtime_Context.Runtime_Fault OR NOT VO_Contract_Valid;
L_Event.Start_Time_MS := VI_System_Time_MS;
L_Event.End_Time_MS := VI_System_Time_MS;
L_Event.Duration_MS := 0;
L_Event.Ordering_Valid := VO_Runtime_Context.DHW_Before_Heating_Valid AND VO_Runtime_Context.State_Publication_Before_Diagnostics_Valid AND VO_Runtime_Context.Output_Projection_Last_Valid;
L_Event.Isolation_Valid := VO_Runtime_Context.Diagnostics_Isolation_Valid AND VO_Runtime_Context.Explainability_Isolation_Valid AND VO_Runtime_Context.Safety_Isolation_Valid AND VO_Runtime_Context.OpenTherm_Ownership_Valid AND VO_Runtime_Context.Cascade_Ownership_Valid;
L_Event.Status_Code := VO_Runtime_Context.Runtime_Status_Code;
L_Event.Status_Text := VO_Runtime_Context.Runtime_Status_Text;
L_Event.Diagnostics_Visible := VO_Runtime_Context.Diagnostics_Isolation_Valid;
L_Event.Explainability_Visible := VO_Runtime_Context.Explainability_Isolation_Valid;
L_Event.Safety_Integrity_Valid := VO_Runtime_Context.Safety_Isolation_Valid;
L_Event.OpenTherm_Ownership_Valid := VO_Runtime_Context.OpenTherm_Ownership_Valid;
L_Event.Cascade_Ownership_Valid := VO_Runtime_Context.Cascade_Ownership_Valid;

fbEventManager(
    VI_Enable := VI_Enable,
    VI_Event := L_Event,
    VIO_Buffer := VO_Runtime_Event_Buffer,
    VO_Event_Stored => L_Event_Stored,
    VO_Buffer_Overflow => L_Buffer_Overflow,
    VO_Manager_Ready => L_Event_Manager_Ready,
    VO_Manager_Status_Code => L_Event_Manager_Code,
    VO_Manager_Status_Text => L_Event_Manager_Text
);

// ======================================================
// SHELL STATUS
// ======================================================
VO_Runtime_Ready := VO_Runtime_Context.Runtime_Ready AND VO_Contract_Valid AND L_Event_Manager_Ready;
VO_Runtime_Fault := VO_Runtime_Context.Runtime_Fault OR NOT VO_Contract_Valid OR L_Buffer_Overflow;

IF VO_Runtime_Fault THEN
    VO_Status_Code := 900;
    VO_Status_Text := 'Heating runtime orchestration shell fault';
ELSIF VO_Runtime_Ready THEN
    VO_Status_Code := 100;
    VO_Status_Text := 'Heating runtime orchestration shell ready';
ELSE
    VO_Status_Code := 10;
    VO_Status_Text := 'Heating runtime orchestration shell active';
END_IF;

END_FUNCTION_BLOCK
// >>> BULK_SYNC_ANCHOR: FB_Heating_Runtime_Orchestration_Shell <<<

(* ---- FB_Heating_Runtime_OT_Instability_Predictor.st ---- *)
// ==============================================================================
// Heating runtime OT instability predictor
// Read-only predictive OT supervision layer.
// ==============================================================================
FUNCTION_BLOCK FB_Heating_Runtime_OT_Instability_Predictor
VAR_INPUT
    VI_Enable : BOOL;
    VI_OT_Degraded : BOOL;
    VI_OT_Command_Valid : BOOL;
END_VAR
VAR_OUTPUT
    VO_OT_Instability_Risk : UINT;
    VO_OT_Degraded_Trend : BOOL;

    VO_Status_Code : UINT;
    VO_Status_Text : STRING(128);
END_VAR

VO_OT_Instability_Risk := 0;
VO_OT_Degraded_Trend := FALSE;

VO_Status_Code := 0;
VO_Status_Text := 'Heating runtime OT predictor disabled';

IF NOT VI_Enable THEN
    RETURN;
END_IF;

IF NOT VI_OT_Command_Valid THEN
    VO_OT_Instability_Risk := 100;
    VO_OT_Degraded_Trend := TRUE;

    VO_Status_Code := 900;
    VO_Status_Text := 'Heating runtime OT instability critical';

ELSIF VI_OT_Degraded THEN
    VO_OT_Instability_Risk := 60;
    VO_OT_Degraded_Trend := TRUE;

    VO_Status_Code := 200;
    VO_Status_Text := 'Heating runtime OT degradation trend';

ELSE
    VO_OT_Instability_Risk := 5;

    VO_Status_Code := 1;
    VO_Status_Text := 'Heating runtime OT nominal';
END_IF;

END_FUNCTION_BLOCK
// >>> BULK_SYNC_ANCHOR: FB_Heating_Runtime_OT_Instability_Predictor <<<

(* ---- FB_Heating_Runtime_Phase_Transition_Observer.st ---- *)
// ==============================================================================
// Heating runtime phase transition observer
// Read-only phase-aware runtime observation layer.
// ==============================================================================
FUNCTION_BLOCK FB_Heating_Runtime_Phase_Transition_Observer
VAR_INPUT
    VI_Enable : BOOL;
    VI_Current_Phase : E_Heating_Runtime_Phase;
    VI_System_Time_MS : UDINT;
END_VAR
VAR_OUTPUT
    VO_Transition : ST_Heating_Runtime_Phase_Transition;
END_VAR
VAR
    L_Previous_Phase : E_Heating_Runtime_Phase;
    L_Transition_Start_MS : UDINT;
END_VAR

VO_Transition.Transition_Active := FALSE;
VO_Transition.Transition_Completed := FALSE;
VO_Transition.Transition_Failed := FALSE;
VO_Transition.Status_Code := 0;
VO_Transition.Status_Text := 'Phase transition observer disabled';

IF NOT VI_Enable THEN
    RETURN;
END_IF;

IF VI_Current_Phase <> L_Previous_Phase THEN

    VO_Transition.Previous_Phase := L_Previous_Phase;
    VO_Transition.Current_Phase := VI_Current_Phase;
    VO_Transition.Next_Phase := VI_Current_Phase;

    VO_Transition.Transition_Active := TRUE;
    VO_Transition.Transition_Completed := TRUE;
    VO_Transition.Transition_Failed := FALSE;

    L_Transition_Start_MS := VI_System_Time_MS;

    VO_Transition.Transition_Start_MS := L_Transition_Start_MS;
    VO_Transition.Transition_End_MS := VI_System_Time_MS;
    VO_Transition.Transition_Duration_MS :=
        VI_System_Time_MS - L_Transition_Start_MS;

    VO_Transition.Sequencing_Valid := TRUE;
    VO_Transition.Ownership_Valid := TRUE;
    VO_Transition.Synchronization_Valid := TRUE;

    VO_Transition.Status_Code := 1;
    VO_Transition.Status_Text := 'Heating runtime phase transition observed';

    L_Previous_Phase := VI_Current_Phase;
END_IF;

END_FUNCTION_BLOCK
// >>> BULK_SYNC_ANCHOR: FB_Heating_Runtime_Phase_Transition_Observer <<<

(* ---- FB_Heating_Runtime_Predictive_Correlation_Weighting_Engine.st ---- *)
// ==============================================================================
// Heating runtime predictive correlation weighting engine
// Read-only predictive adaptive correlation layer.
// ==============================================================================
FUNCTION_BLOCK FB_Heating_Runtime_Predictive_Correlation_Weighting_Engine
VAR_INPUT
    VI_Enable : BOOL;
    VI_Runtime_Risk : UINT;
    VI_Cascade_Risk : UINT;
    VI_OT_Risk : UINT;
END_VAR
VAR_OUTPUT
    VO_Correlation_Score : UINT;
    VO_Correlation_Degraded : BOOL;

    VO_Status_Code : UINT;
    VO_Status_Text : STRING(128);
END_VAR
VAR
    L_Total : UDINT;
END_VAR

VO_Correlation_Score := 0;
VO_Correlation_Degraded := FALSE;

VO_Status_Code := 0;
VO_Status_Text := 'Heating predictive correlation engine disabled';

IF NOT VI_Enable THEN
    RETURN;
END_IF;

// ======================================================
// SAFE ARITHMETIC
// ======================================================
L_Total :=
    TO_UDINT(VI_Runtime_Risk) +
    TO_UDINT(VI_Cascade_Risk) +
    TO_UDINT(VI_OT_Risk);

VO_Correlation_Score :=
    TO_UINT(L_Total / 3);

// ======================================================
// CORRELATION ANALYSIS
// ======================================================
IF VO_Correlation_Score > 70 THEN
    VO_Correlation_Degraded := TRUE;

    VO_Status_Code := 900;
    VO_Status_Text := 'Heating predictive correlation critical';

ELSIF VO_Correlation_Score > 40 THEN
    VO_Correlation_Degraded := TRUE;

    VO_Status_Code := 200;
    VO_Status_Text := 'Heating predictive correlation degraded';

ELSE
    VO_Status_Code := 1;
    VO_Status_Text := 'Heating predictive correlation nominal';
END_IF;

END_FUNCTION_BLOCK
// >>> BULK_SYNC_ANCHOR: FB_Heating_Runtime_Predictive_Correlation_Weighting_Engine <<<

(* ---- FB_Heating_Runtime_RootCause_Correlator.st ---- *)
// ==============================================================================
// Heating runtime root-cause correlator
// Read-only runtime causality correlation layer.
// ==============================================================================
FUNCTION_BLOCK FB_Heating_Runtime_RootCause_Correlator
VAR_INPUT
    VI_Enable : BOOL;
    VI_Anomaly : ST_Heating_Runtime_Anomaly;
END_VAR
VAR_OUTPUT
    VO_Node : ST_Heating_Runtime_Causality_Node;
END_VAR

VO_Node.Node_Active := FALSE;
VO_Node.Root_Cause_Candidate := FALSE;
VO_Node.Runtime_Degraded := FALSE;
VO_Node.Runtime_Fault := FALSE;

VO_Node.Cascade_Degraded := FALSE;
VO_Node.Cascade_Boiler_Loss := FALSE;

VO_Node.OpenTherm_Degraded := FALSE;
VO_Node.OpenTherm_Command_Invalid := FALSE;

VO_Node.Diagnostics_Degraded := FALSE;
VO_Node.Explainability_Degraded := FALSE;

VO_Node.Sequencing_Invalid := FALSE;
VO_Node.Ownership_Invalid := FALSE;
VO_Node.Synchronization_Invalid := FALSE;

VO_Node.Severity_Level := 0;

VO_Node.Status_Code := 0;
VO_Node.Status_Text := 'Heating runtime root-cause correlator disabled';

IF NOT VI_Enable THEN
    RETURN;
END_IF;

VO_Node.Node_Active := VI_Anomaly.Anomaly_Active;

VO_Node.Runtime_Degraded := VI_Anomaly.Runtime_Degraded;
VO_Node.Runtime_Fault :=
    VI_Anomaly.Critical_Anomaly;

VO_Node.Cascade_Degraded :=
    VI_Anomaly.Cascade_Degraded;

VO_Node.Cascade_Boiler_Loss :=
    VI_Anomaly.Cascade_Boiler_Loss_Detected;

VO_Node.OpenTherm_Degraded :=
    VI_Anomaly.OpenTherm_Transport_Degraded;

VO_Node.OpenTherm_Command_Invalid :=
    VI_Anomaly.OpenTherm_Command_Invalid;

VO_Node.Diagnostics_Degraded :=
    VI_Anomaly.Diagnostics_Degraded;

VO_Node.Explainability_Degraded :=
    VI_Anomaly.Explainability_Degraded;

VO_Node.Sequencing_Invalid :=
    VI_Anomaly.Sequencing_Invalid;

VO_Node.Ownership_Invalid :=
    VI_Anomaly.Ownership_Invalid;

VO_Node.Synchronization_Invalid :=
    VI_Anomaly.Synchronization_Invalid;

VO_Node.Severity_Level :=
    VI_Anomaly.Severity_Level;

VO_Node.Root_Cause_Candidate :=
    VI_Anomaly.Critical_Anomaly OR
    VI_Anomaly.Sequencing_Invalid OR
    VI_Anomaly.Ownership_Invalid OR
    VI_Anomaly.Synchronization_Invalid;

IF VO_Node.Root_Cause_Candidate THEN
    VO_Node.Status_Code := 900;
    VO_Node.Status_Text := 'Heating runtime root-cause candidate detected';
ELSE
    VO_Node.Status_Code := 1;
    VO_Node.Status_Text := 'Heating runtime causality nominal';
END_IF;

END_FUNCTION_BLOCK
// >>> BULK_SYNC_ANCHOR: FB_Heating_Runtime_RootCause_Correlator <<<

(* ---- FB_Heating_Runtime_Stability_Model.st ---- *)
// ==============================================================================
// Heating runtime stability model
// Read-only predictive runtime stability layer.
// ==============================================================================
FUNCTION_BLOCK FB_Heating_Runtime_Stability_Model
VAR_INPUT
    VI_Enable : BOOL;
    VI_Runtime_Degraded : BOOL;
    VI_Runtime_Critical : BOOL;
END_VAR
VAR_OUTPUT
    VO_Runtime_Stable : BOOL;
    VO_Stability_Score : UINT;

    VO_Status_Code : UINT;
    VO_Status_Text : STRING(128);
END_VAR

VO_Runtime_Stable := FALSE;
VO_Stability_Score := 0;

VO_Status_Code := 0;
VO_Status_Text := 'Heating runtime stability model disabled';

IF NOT VI_Enable THEN
    RETURN;
END_IF;

IF VI_Runtime_Critical THEN
    VO_Runtime_Stable := FALSE;
    VO_Stability_Score := 0;

    VO_Status_Code := 900;
    VO_Status_Text := 'Heating runtime critically unstable';

ELSIF VI_Runtime_Degraded THEN
    VO_Runtime_Stable := FALSE;
    VO_Stability_Score := 50;

    VO_Status_Code := 200;
    VO_Status_Text := 'Heating runtime degraded stability';

ELSE
    VO_Runtime_Stable := TRUE;
    VO_Stability_Score := 100;

    VO_Status_Code := 1;
    VO_Status_Text := 'Heating runtime stable';
END_IF;

END_FUNCTION_BLOCK
// >>> BULK_SYNC_ANCHOR: FB_Heating_Runtime_Stability_Model <<<

(* ---- FB_Heating_Runtime_State_Publication_Phase.st ---- *)
// ==============================================================================
// Heating runtime state publication phase
// Owns publication of finalized runtime outputs into global state/status layers.
// Does NOT calculate heating logic and does NOT mutate outputs.
// ==============================================================================
FUNCTION_BLOCK FB_Heating_Runtime_State_Publication_Phase
VAR_INPUT
    VI_Enable : BOOL;
    VI_Zone_Valves : ARRAY[1..GVL_CONSTANTS.C_MAX_HEATING_CIRCUITS] OF BOOL;
    VI_Manifold_Pumps : ARRAY[1..GVL_CONSTANTS.C_MAX_MANIFOLDS] OF BOOL;
    VI_Manifold_Valves : ARRAY[1..GVL_CONSTANTS.C_MAX_MANIFOLDS] OF REAL;
    VI_Boiler_OT_Enable : ARRAY[1..GVL_CONSTANTS.C_MAX_BOILERS] OF BOOL;
    VI_Boiler_OT_Setpoint : ARRAY[1..GVL_CONSTANTS.C_MAX_BOILERS] OF REAL;
    VI_Backup_Circulation_Pump : BOOL;
    VI_Electric_Heater_Enable : BOOL;
    VI_Freeze_Risk_Status : BOOL;
    VI_Manifold_Status : ARRAY[1..GVL_CONSTANTS.C_MAX_MANIFOLDS] OF ST_Manifold_Status;
    VI_Boiler_Status : ARRAY[1..GVL_CONSTANTS.C_MAX_BOILERS] OF ST_Boiler_Status;
    VI_DHW_Heating_Pump : BOOL;
    VI_DHW_Circ_Pump : BOOL;
    VI_DHW_Status : ST_DHW_Status;
END_VAR
VAR_OUTPUT
    VO_Executed : BOOL;
    VO_Valid : BOOL;
END_VAR
VAR
    L_i : INT;
END_VAR

VO_Executed := FALSE;
VO_Valid := FALSE;

IF NOT VI_Enable THEN
    RETURN;
END_IF;

FOR L_i := 1 TO GVL_CONSTANTS.C_MAX_HEATING_CIRCUITS DO
    GVL_STATE.G_Zone_Valves[L_i] := VI_Zone_Valves[L_i];
END_FOR;

FOR L_i := 1 TO GVL_CONSTANTS.C_MAX_MANIFOLDS DO
    GVL_STATE.G_Manifold_Pumps[L_i] := VI_Manifold_Pumps[L_i];
    GVL_STATE.G_Manifold_Valves[L_i] := VI_Manifold_Valves[L_i];
    GVL_STATUS.G_Manifold_Status[L_i] := VI_Manifold_Status[L_i];
END_FOR;

FOR L_i := 1 TO GVL_CONSTANTS.C_MAX_BOILERS DO
    GVL_STATE.G_Boiler_OT_Enable[L_i] := VI_Boiler_OT_Enable[L_i];
    GVL_STATE.G_Boiler_OT_Setpoint[L_i] := VI_Boiler_OT_Setpoint[L_i];
    GVL_STATUS.G_Boiler_Status[L_i] := VI_Boiler_Status[L_i];
END_FOR;

GVL_STATE.G_Backup_Circulation_Pump := VI_Backup_Circulation_Pump;
GVL_STATE.G_Electric_Heater_Enable := VI_Electric_Heater_Enable;
GVL_STATE.G_Safety_Freeze_Risk := VI_Freeze_Risk_Status;
GVL_STATE.G_DHW_Heating_Pump := VI_DHW_Heating_Pump;
GVL_STATE.G_DHW_Circ_Pump := VI_DHW_Circ_Pump;
GVL_STATUS.G_DHW_Status := VI_DHW_Status;

VO_Executed := TRUE;
VO_Valid := TRUE;

END_FUNCTION_BLOCK
// >>> BULK_SYNC_ANCHOR: FB_Heating_Runtime_State_Publication_Phase <<<

(* ---- FB_Heating_Runtime_Supervision_Confidence_Analyzer.st ---- *)
// ==============================================================================
// Heating runtime supervision confidence analyzer
// Read-only adaptive confidence supervision layer.
// ==============================================================================
FUNCTION_BLOCK FB_Heating_Runtime_Supervision_Confidence_Analyzer
VAR_INPUT
    VI_Enable : BOOL;
    VI_Runtime_Stable : BOOL;
    VI_Runtime_Degraded : BOOL;
END_VAR
VAR_OUTPUT
    VO_Supervision_Confidence : UINT;
    VO_Confidence_Degraded : BOOL;

    VO_Status_Code : UINT;
    VO_Status_Text : STRING(128);
END_VAR

VO_Supervision_Confidence := 0;
VO_Confidence_Degraded := FALSE;

VO_Status_Code := 0;
VO_Status_Text := 'Heating supervision confidence analyzer disabled';

IF NOT VI_Enable THEN
    RETURN;
END_IF;

IF VI_Runtime_Degraded THEN
    VO_Supervision_Confidence := 40;
    VO_Confidence_Degraded := TRUE;

    VO_Status_Code := 200;
    VO_Status_Text := 'Heating supervision confidence degraded';

ELSIF VI_Runtime_Stable THEN
    VO_Supervision_Confidence := 95;

    VO_Status_Code := 1;
    VO_Status_Text := 'Heating supervision confidence nominal';

ELSE
    VO_Supervision_Confidence := 60;

    VO_Status_Code := 100;
    VO_Status_Text := 'Heating supervision confidence transitional';
END_IF;

END_FUNCTION_BLOCK
// >>> BULK_SYNC_ANCHOR: FB_Heating_Runtime_Supervision_Confidence_Analyzer <<<

(* ---- FB_Heating_Runtime_Supervisory_Enrichment.st ---- *)
// ==============================================================================
// Heating runtime supervisory enrichment
// Passive observability-only connector for restored supervisory FB stack.
//
// DOES NOT own runtime.
// DOES NOT own heating logic.
// DOES NOT own diagnostics authority.
// DOES NOT own OpenTherm transport.
// DOES NOT write outputs or commands.
// ==============================================================================
FUNCTION_BLOCK FB_Heating_Runtime_Supervisory_Enrichment
VAR_INPUT
    VI_Enable : BOOL;
    VI_System_Time_MS : UDINT;
    VI_Runtime_Context : ST_Heating_Runtime_Context;
    VI_Phase_Event : ST_Heating_Runtime_Phase_Event;
    VI_Anomaly : ST_Heating_Runtime_Anomaly;
    VI_Cascade_Boiler_Count : UINT;
    VI_OT_Command_Valid : BOOL;
END_VAR
VAR_IN_OUT
    VIO_Event_Buffer : ST_Heating_Runtime_Event_Buffer;
    VIO_Execution_Timeline : ST_Heating_Runtime_Execution_Timeline;
END_VAR
VAR_OUTPUT
    VO_Causality_Node : ST_Heating_Runtime_Causality_Node;
    VO_Causality_Edge : ST_Heating_Runtime_Causality_Edge;
    VO_Blackbox_Event : ST_Heating_Runtime_Blackbox_Event;
    VO_Predictive_State : ST_Heating_Runtime_Predictive_State;
    VO_Status_Code : UINT;
    VO_Status_Text : STRING(128);
END_VAR
VAR
    fbEventManager : FB_Heating_Runtime_Event_Manager;
    fbTimelineObserver : FB_Heating_Runtime_Timeline_Observer;
    fbRootCauseCorrelator : FB_Heating_Runtime_RootCause_Correlator;
    fbReconstructionEngine : FB_Heating_Runtime_Event_Reconstruction_Engine;
    fbStabilityModel : FB_Heating_Runtime_Stability_Model;
    fbOTCascadeCorrelator : FB_Heating_Runtime_OT_Cascade_Correlator;
    fbOTInstabilityPredictor : FB_Heating_Runtime_OT_Instability_Predictor;
    fbPredictiveCorrelation : FB_Heating_Runtime_Predictive_Correlation_Weighting_Engine;

    L_Frame : ST_Heating_Runtime_Execution_Frame;
    L_Runtime_Risk : UINT;
    L_Cascade_Risk : UINT;
    L_Circuit_i : INT;
    L_Circuit_Event_Active : BOOL;
    L_Circuit_Event_Code : UINT;
    L_Circuit_Event_Text : STRING(128);
    L_Phase_Event : ST_Heating_Runtime_Phase_Event;
    L_Anomaly : ST_Heating_Runtime_Anomaly;
END_VAR

// ======================================================
// DEFAULTS
// ======================================================
VO_Status_Code := 0;
VO_Status_Text := 'Heating runtime supervisory enrichment disabled';

IF NOT VI_Enable THEN
    RETURN;
END_IF;

// ======================================================
// PASSIVE CIRCUIT EDGE INGESTION
// ======================================================
// Circuit control publishes edge flags only. This supervisory connector is the
// integration boundary that raises those passive edges into the event/anomaly
// stream used by timeline, reconstruction and causality observers.
L_Phase_Event := VI_Phase_Event;
L_Anomaly := VI_Anomaly;
L_Circuit_Event_Active := FALSE;
L_Circuit_Event_Code := 0;
L_Circuit_Event_Text := '';

FOR L_Circuit_i := 1 TO GVL_CONSTANTS.C_MAX_HEATING_CIRCUITS DO
    IF GVL_Heating_Circuit_Explainability.G_Source_Loss_Event[L_Circuit_i] THEN
        L_Circuit_Event_Active := TRUE;
        L_Circuit_Event_Code := 804;
        L_Circuit_Event_Text := 'Heating circuit temperature source loss';
        EXIT;
    ELSIF GVL_Heating_Circuit_Explainability.G_Fallback_Activated_Event[L_Circuit_i] THEN
        L_Circuit_Event_Active := TRUE;
        L_Circuit_Event_Code := 802;
        L_Circuit_Event_Text := 'Heating circuit fallback activated';
        EXIT;
    ELSIF GVL_Heating_Circuit_Explainability.G_Fallback_Recovered_Event[L_Circuit_i] THEN
        L_Circuit_Event_Active := TRUE;
        L_Circuit_Event_Code := 803;
        L_Circuit_Event_Text := 'Heating circuit fallback recovered';
        EXIT;
    ELSIF GVL_Heating_Circuit_Explainability.G_Source_Switched_Event[L_Circuit_i] THEN
        L_Circuit_Event_Active := TRUE;
        L_Circuit_Event_Code := 801;
        L_Circuit_Event_Text := 'Heating circuit temperature source switched';
        EXIT;
    END_IF;
END_FOR;

IF L_Circuit_Event_Active THEN
    L_Phase_Event.Phase := VI_Runtime_Context.Current_Phase;
    L_Phase_Event.Event_Active := TRUE;
    L_Phase_Event.Event_Completed := TRUE;
    L_Phase_Event.Event_Failed := FALSE;
    L_Phase_Event.Start_Time_MS := VI_System_Time_MS;
    L_Phase_Event.End_Time_MS := VI_System_Time_MS;
    L_Phase_Event.Duration_MS := 0;
    L_Phase_Event.Ordering_Valid := TRUE;
    L_Phase_Event.Isolation_Valid := TRUE;
    L_Phase_Event.Status_Code := L_Circuit_Event_Code;
    L_Phase_Event.Status_Text := L_Circuit_Event_Text;
    L_Phase_Event.Diagnostics_Visible := TRUE;
    L_Phase_Event.Explainability_Visible := TRUE;
    L_Phase_Event.Safety_Integrity_Valid := TRUE;
    L_Phase_Event.OpenTherm_Ownership_Valid := TRUE;
    L_Phase_Event.Cascade_Ownership_Valid := TRUE;

    L_Anomaly.Anomaly_Active := TRUE;
    L_Anomaly.Runtime_Degraded := L_Anomaly.Runtime_Degraded OR (L_Circuit_Event_Code = 802) OR (L_Circuit_Event_Code = 804);
    L_Anomaly.Diagnostics_Degraded := L_Anomaly.Diagnostics_Degraded OR (L_Circuit_Event_Code = 804);
    L_Anomaly.Explainability_Degraded := L_Anomaly.Explainability_Degraded OR (L_Circuit_Event_Code = 804);

    IF L_Circuit_Event_Code = 804 THEN
        IF L_Anomaly.Severity_Level < 80 THEN
            L_Anomaly.Severity_Level := 80;
        END_IF;
        L_Anomaly.Status_Code := 804;
        L_Anomaly.Status_Text := 'Heating circuit source loss observed';
    ELSIF L_Circuit_Event_Code = 802 THEN
        IF L_Anomaly.Severity_Level < 40 THEN
            L_Anomaly.Severity_Level := 40;
        END_IF;
        L_Anomaly.Status_Code := 802;
        L_Anomaly.Status_Text := 'Heating circuit fallback activation observed';
    ELSIF L_Circuit_Event_Code = 803 THEN
        L_Anomaly.Status_Code := 803;
        L_Anomaly.Status_Text := 'Heating circuit fallback recovery observed';
    ELSE
        L_Anomaly.Status_Code := 801;
        L_Anomaly.Status_Text := 'Heating circuit source switch observed';
    END_IF;
END_IF;

// ======================================================
// EXECUTION FRAME FROM CURRENT RUNTIME CONTEXT
// ======================================================
L_Frame.Phase := VI_Runtime_Context.Current_Phase;
L_Frame.Frame_Started := TRUE;
L_Frame.Frame_Completed := VI_Runtime_Context.Output_Projection_Executed;
L_Frame.Frame_Failed := VI_Runtime_Context.Runtime_Fault;
L_Frame.Frame_Start_MS := VI_System_Time_MS;
L_Frame.Frame_End_MS := VI_System_Time_MS;
L_Frame.Frame_Duration_MS := 0;

L_Frame.Sequencing_Valid :=
    VI_Runtime_Context.DHW_Before_Heating_Valid AND
    VI_Runtime_Context.State_Publication_Before_Diagnostics_Valid AND
    VI_Runtime_Context.Output_Projection_Last_Valid;

L_Frame.Ownership_Valid :=
    VI_Runtime_Context.OpenTherm_Ownership_Valid AND
    VI_Runtime_Context.Cascade_Ownership_Valid AND
    VI_Runtime_Context.Safety_Isolation_Valid;

L_Frame.Synchronization_Valid :=
    VI_Runtime_Context.Diagnostics_Isolation_Valid AND
    VI_Runtime_Context.Explainability_Isolation_Valid;

L_Frame.Runtime_Jitter_Detected := L_Anomaly.Runtime_Jitter_Detected;
L_Frame.Runtime_Latency_Detected := L_Anomaly.Runtime_Latency_Detected;
L_Frame.Runtime_Degraded := L_Anomaly.Runtime_Degraded;
L_Frame.Status_Code := VI_Runtime_Context.Runtime_Status_Code;
L_Frame.Status_Text := VI_Runtime_Context.Runtime_Status_Text;

fbTimelineObserver(
    VI_Enable := TRUE,
    VI_Frame := L_Frame,
    VIO_Timeline := VIO_Execution_Timeline
);

// ======================================================
// EVENT BUFFER
// ======================================================
fbEventManager(
    VI_Enable := TRUE,
    VI_Event := L_Phase_Event,
    VIO_Buffer := VIO_Event_Buffer
);

// ======================================================
// ROOT-CAUSE / CAUSALITY NODE
// ======================================================
fbRootCauseCorrelator(
    VI_Enable := TRUE,
    VI_Anomaly := L_Anomaly
);

VO_Causality_Node := fbRootCauseCorrelator.VO_Node;

// ======================================================
// CAUSALITY EDGE BUILT FROM NODE STATE
// ======================================================
VO_Causality_Edge.Source_Node_ID := 1;
VO_Causality_Edge.Target_Node_ID := 2;
VO_Causality_Edge.Edge_Active := VO_Causality_Node.Node_Active;
VO_Causality_Edge.Propagation_Detected :=
    VO_Causality_Node.Runtime_Degraded OR
    VO_Causality_Node.Runtime_Fault OR
    VO_Causality_Node.Cascade_Degraded OR
    VO_Causality_Node.OpenTherm_Degraded OR
    VO_Causality_Node.Sequencing_Invalid OR
    VO_Causality_Node.Ownership_Invalid OR
    VO_Causality_Node.Synchronization_Invalid;

VO_Causality_Edge.Runtime_Propagation :=
    VO_Causality_Node.Runtime_Degraded OR VO_Causality_Node.Runtime_Fault;
VO_Causality_Edge.Cascade_Propagation := VO_Causality_Node.Cascade_Degraded;
VO_Causality_Edge.OpenTherm_Propagation := VO_Causality_Node.OpenTherm_Degraded;
VO_Causality_Edge.Diagnostics_Propagation := VO_Causality_Node.Diagnostics_Degraded;
VO_Causality_Edge.Sequencing_Propagation := VO_Causality_Node.Sequencing_Invalid;
VO_Causality_Edge.Ownership_Propagation := VO_Causality_Node.Ownership_Invalid;
VO_Causality_Edge.Synchronization_Propagation := VO_Causality_Node.Synchronization_Invalid;
VO_Causality_Edge.Severity_Level := VO_Causality_Node.Severity_Level;
VO_Causality_Edge.Critical_Path := VO_Causality_Node.Root_Cause_Candidate;
VO_Causality_Edge.Status_Code := VO_Causality_Node.Status_Code;
VO_Causality_Edge.Status_Text := VO_Causality_Node.Status_Text;

// ======================================================
// FORENSIC RECONSTRUCTION
// ======================================================
fbReconstructionEngine(
    VI_Enable := TRUE,
    VI_Node := VO_Causality_Node,
    VI_Edge := VO_Causality_Edge,
    VI_System_Time_MS := VI_System_Time_MS
);

VO_Blackbox_Event := fbReconstructionEngine.VO_Event;

// ======================================================
// STABILITY / OT / CASCADE PREDICTIVE SUPERVISION
// ======================================================
fbStabilityModel(
    VI_Enable := TRUE,
    VI_Runtime_Degraded := L_Anomaly.Runtime_Degraded,
    VI_Runtime_Critical := L_Anomaly.Critical_Anomaly
);

fbOTCascadeCorrelator(
    VI_Enable := TRUE,
    VI_Cascade_Degraded := L_Anomaly.Cascade_Degraded,
    VI_OT_Degraded := L_Anomaly.OpenTherm_Transport_Degraded,
    VI_OT_Command_Valid := VI_OT_Command_Valid,
    VI_Boiler_Count := VI_Cascade_Boiler_Count
);

fbOTInstabilityPredictor(
    VI_Enable := TRUE,
    VI_OT_Degraded := L_Anomaly.OpenTherm_Transport_Degraded,
    VI_OT_Command_Valid := VI_OT_Command_Valid
);

IF L_Anomaly.Critical_Anomaly THEN
    L_Runtime_Risk := 100;
ELSIF L_Anomaly.Runtime_Degraded THEN
    L_Runtime_Risk := 60;
ELSE
    L_Runtime_Risk := 0;
END_IF;

IF L_Anomaly.Cascade_Boiler_Loss_Detected THEN
    L_Cascade_Risk := 100;
ELSIF L_Anomaly.Cascade_Degraded THEN
    L_Cascade_Risk := 60;
ELSE
    L_Cascade_Risk := 0;
END_IF;

fbPredictiveCorrelation(
    VI_Enable := TRUE,
    VI_Runtime_Risk := L_Runtime_Risk,
    VI_Cascade_Risk := L_Cascade_Risk,
    VI_OT_Risk := fbOTInstabilityPredictor.VO_OT_Instability_Risk
);

// ======================================================
// PREDICTIVE PUBLICATION MODEL
// ======================================================
VO_Predictive_State.Predictive_Analytics_Visible := TRUE;
VO_Predictive_State.Predictive_Analytics_Degraded := fbPredictiveCorrelation.VO_Correlation_Degraded;
VO_Predictive_State.Predictive_Analytics_Attention := fbPredictiveCorrelation.VO_Correlation_Score > 40;
VO_Predictive_State.Runtime_Stable := fbStabilityModel.VO_Runtime_Stable;
VO_Predictive_State.Runtime_Stability_Score := fbStabilityModel.VO_Stability_Score;
VO_Predictive_State.Runtime_Degradation_Observation := L_Runtime_Risk;
VO_Predictive_State.Runtime_Failure_Observation := SEL(L_Anomaly.Critical_Anomaly, 0, 100);
VO_Predictive_State.Cascade_Degradation_Observation := L_Cascade_Risk;
VO_Predictive_State.Cascade_Degraded_Trend_Visible := fbOTCascadeCorrelator.VO_Correlation_Detected;
VO_Predictive_State.OpenTherm_Instability_Observation := fbOTInstabilityPredictor.VO_OT_Instability_Risk;
VO_Predictive_State.OpenTherm_Degraded_Trend_Visible := fbOTInstabilityPredictor.VO_OT_Degraded_Trend;
VO_Predictive_State.Sequencing_Observation := SEL(VO_Causality_Node.Sequencing_Invalid, 0, 100);
VO_Predictive_State.Ownership_Observation := SEL(VO_Causality_Node.Ownership_Invalid, 0, 100);
VO_Predictive_State.Synchronization_Observation := SEL(VO_Causality_Node.Synchronization_Invalid, 0, 100);
VO_Predictive_State.Status_Code := fbPredictiveCorrelation.VO_Status_Code;
VO_Predictive_State.Status_Text := fbPredictiveCorrelation.VO_Status_Text;

VO_Status_Code := fbPredictiveCorrelation.VO_Status_Code;
VO_Status_Text := fbPredictiveCorrelation.VO_Status_Text;

END_FUNCTION_BLOCK
// >>> BULK_SYNC_ANCHOR: FB_Heating_Runtime_Supervisory_Enrichment <<<

(* ---- FB_Heating_Runtime_Supervisory_Publication_Adapter.st ---- *)
// ==============================================================================
// Heating runtime supervisory publication adapter
//
// Canonical supervisory publication adapter.
//
// Consolidates predictive, causality, explainability and reconstruction
// semantics into a single passive supervisory publication surface.
//
// DOES NOT own runtime authority.
// DOES NOT own outputs.
// DOES NOT modify runtime execution.
// ==============================================================================
FUNCTION_BLOCK FB_Heating_Runtime_Supervisory_Publication_Adapter
VAR_INPUT
    VI_Enable : BOOL;

    VI_Predictive_State : ST_Heating_Runtime_Predictive_State;
    VI_Causality_Node : ST_Heating_Runtime_Causality_Node;
    VI_Causality_Edge : ST_Heating_Runtime_Causality_Edge;
    VI_Blackbox_Event : ST_Heating_Runtime_Blackbox_Event;
    VI_Anomaly : ST_Heating_Runtime_Anomaly;
END_VAR

IF NOT VI_Enable THEN
    RETURN;
END_IF;

GVL_Heating_Runtime_Supervisory_Publication.G_Publication.Supervisory_Visible := TRUE;

// ======================================================
// PREDICTIVE
// ======================================================
GVL_Heating_Runtime_Supervisory_Publication.G_Publication.Predictive_State :=
    VI_Predictive_State;

GVL_Heating_Runtime_Supervisory_Publication.G_Publication.Source_Instability_Attention :=
    VI_Predictive_State.Source_Instability_Attention;

GVL_Heating_Runtime_Supervisory_Publication.G_Publication.Source_Oscillation_Trend_Visible :=
    VI_Predictive_State.Source_Oscillation_Trend_Visible;

// ======================================================
// RUNTIME / DEGRADATION
// ======================================================
GVL_Heating_Runtime_Supervisory_Publication.G_Publication.Runtime_Degraded :=
    VI_Anomaly.Runtime_Degraded;

GVL_Heating_Runtime_Supervisory_Publication.G_Publication.Runtime_Fault :=
    VI_Anomaly.Critical_Anomaly;

GVL_Heating_Runtime_Supervisory_Publication.G_Publication.Explainability_Degraded :=
    VI_Anomaly.Explainability_Degraded;

GVL_Heating_Runtime_Supervisory_Publication.G_Publication.Diagnostics_Degraded :=
    VI_Anomaly.Diagnostics_Degraded;

// ======================================================
// CAUSALITY
// ======================================================
GVL_Heating_Runtime_Supervisory_Publication.G_Publication.Causality_Active :=
    VI_Causality_Node.Node_Active;

GVL_Heating_Runtime_Supervisory_Publication.G_Publication.Propagation_Detected :=
    VI_Causality_Edge.Propagation_Detected;

// ======================================================
// RECONSTRUCTION
// ======================================================
GVL_Heating_Runtime_Supervisory_Publication.G_Publication.Reconstruction_Visible :=
    VI_Blackbox_Event.Event_Visible;

// ======================================================
// STATUS
// ======================================================
GVL_Heating_Runtime_Supervisory_Publication.G_Publication.Status_Code :=
    VI_Predictive_State.Status_Code;

GVL_Heating_Runtime_Supervisory_Publication.G_Publication.Status_Text :=
    VI_Predictive_State.Status_Text;

END_FUNCTION_BLOCK
// >>> BULK_SYNC_ANCHOR: FB_Heating_Runtime_Supervisory_Publication_Adapter <<<

(* ---- FB_Heating_Runtime_Synchronization_Monitor.st ---- *)
// ==============================================================================
// Heating runtime synchronization monitor
// Read-only orchestration synchronization layer.
// DOES NOT own runtime.
// DOES NOT own heating logic.
// DOES NOT own diagnostics.
// DOES NOT own OpenTherm transport.
// DOES NOT migrate runtime ownership.
// ==============================================================================
FUNCTION_BLOCK FB_Heating_Runtime_Synchronization_Monitor
VAR_INPUT
    VI_Enable : BOOL;
    VI_Context : ST_Heating_Runtime_Context;
    VI_Bridge : ST_Heating_Runtime_Integration_Bridge;
END_VAR
VAR_OUTPUT
    VO_Synchronized : BOOL;
    VO_Phase_Synchronized : BOOL;
    VO_Ownership_Synchronized : BOOL;
    VO_Sequencing_Synchronized : BOOL;

    VO_Status_Code : UINT;
    VO_Status_Text : STRING(128);
END_VAR
VAR
    L_Phase_Valid : BOOL;
    L_Ownership_Valid : BOOL;
    L_Sequencing_Valid : BOOL;
END_VAR

// ======================================================
// DEFAULTS
// ======================================================
VO_Synchronized := FALSE;
VO_Phase_Synchronized := FALSE;
VO_Ownership_Synchronized := FALSE;
VO_Sequencing_Synchronized := FALSE;

VO_Status_Code := 0;
VO_Status_Text := 'Heating runtime synchronization monitor disabled';

L_Phase_Valid := TRUE;
L_Ownership_Valid := TRUE;
L_Sequencing_Valid := TRUE;

IF NOT VI_Enable THEN
    RETURN;
END_IF;

// ======================================================
// PHASE SYNCHRONIZATION
// ======================================================
IF VI_Context.Current_Phase <> VI_Bridge.Current_Phase THEN
    L_Phase_Valid := FALSE;
END_IF;

IF NOT VI_Bridge.Runtime_Synchronized THEN
    L_Phase_Valid := FALSE;
END_IF;

// ======================================================
// OWNERSHIP SYNCHRONIZATION
// ======================================================
IF NOT VI_Bridge.Runtime_Ownership_Valid THEN
    L_Ownership_Valid := FALSE;
END_IF;

IF NOT VI_Bridge.Diagnostics_Ownership_Valid THEN
    L_Ownership_Valid := FALSE;
END_IF;

IF NOT VI_Bridge.Explainability_Ownership_Valid THEN
    L_Ownership_Valid := FALSE;
END_IF;

IF NOT VI_Bridge.OpenTherm_Ownership_Valid THEN
    L_Ownership_Valid := FALSE;
END_IF;

IF NOT VI_Bridge.Cascade_Ownership_Valid THEN
    L_Ownership_Valid := FALSE;
END_IF;

IF NOT VI_Bridge.Safety_Ownership_Valid THEN
    L_Ownership_Valid := FALSE;
END_IF;

// ======================================================
// SEQUENCING SYNCHRONIZATION
// ======================================================
IF NOT VI_Bridge.DHW_Before_Heating_Valid THEN
    L_Sequencing_Valid := FALSE;
END_IF;

IF NOT VI_Bridge.Diagnostics_After_Publication_Valid THEN
    L_Sequencing_Valid := FALSE;
END_IF;

IF NOT VI_Bridge.Output_Projection_Last_Valid THEN
    L_Sequencing_Valid := FALSE;
END_IF;

// ======================================================
// OUTPUTS
// ======================================================
VO_Phase_Synchronized := L_Phase_Valid;
VO_Ownership_Synchronized := L_Ownership_Valid;
VO_Sequencing_Synchronized := L_Sequencing_Valid;

VO_Synchronized :=
    L_Phase_Valid AND
    L_Ownership_Valid AND
    L_Sequencing_Valid AND
    VI_Bridge.Runtime_Migration_Allowed;

// ======================================================
// STATUS
// ======================================================
IF NOT L_Phase_Valid THEN
    VO_Status_Code := 100;
    VO_Status_Text := 'Heating runtime phase synchronization failed';

ELSIF NOT L_Ownership_Valid THEN
    VO_Status_Code := 200;
    VO_Status_Text := 'Heating runtime ownership synchronization failed';

ELSIF NOT L_Sequencing_Valid THEN
    VO_Status_Code := 300;
    VO_Status_Text := 'Heating runtime sequencing synchronization failed';

ELSIF NOT VI_Bridge.Runtime_Migration_Allowed THEN
    VO_Status_Code := 400;
    VO_Status_Text := 'Heating runtime migration not allowed';

ELSE
    VO_Status_Code := 1;
    VO_Status_Text := 'Heating runtime synchronization valid';
END_IF;

END_FUNCTION_BLOCK
// >>> BULK_SYNC_ANCHOR: FB_Heating_Runtime_Synchronization_Monitor <<<

(* ---- FB_Heating_Runtime_Timeline_Observer.st ---- *)
// ==============================================================================
// Heating runtime timeline observer
// Read-only deterministic execution timeline layer.
// ==============================================================================
FUNCTION_BLOCK FB_Heating_Runtime_Timeline_Observer
VAR_INPUT
    VI_Enable : BOOL;
    VI_Frame : ST_Heating_Runtime_Execution_Frame;
END_VAR
VAR_IN_OUT
    VIO_Timeline : ST_Heating_Runtime_Execution_Timeline;
END_VAR
VAR
    L_Index : UINT;
END_VAR

IF NOT VI_Enable THEN
    RETURN;
END_IF;

L_Index := VIO_Timeline.Write_Index + 1;

IF L_Index > 64 THEN
    L_Index := 1;
    VIO_Timeline.Timeline_Overflow := TRUE;
END_IF;

VIO_Timeline.Frames[L_Index] := VI_Frame;
VIO_Timeline.Write_Index := L_Index;

IF VIO_Timeline.Frame_Count < 64 THEN
    VIO_Timeline.Frame_Count :=
        VIO_Timeline.Frame_Count + 1;
END_IF;

VIO_Timeline.Sequencing_Valid :=
    VI_Frame.Sequencing_Valid;

VIO_Timeline.Ownership_Valid :=
    VI_Frame.Ownership_Valid;

VIO_Timeline.Synchronization_Valid :=
    VI_Frame.Synchronization_Valid;

VIO_Timeline.Runtime_Jitter_Detected :=
    VI_Frame.Runtime_Jitter_Detected;

VIO_Timeline.Runtime_Latency_Detected :=
    VI_Frame.Runtime_Latency_Detected;

VIO_Timeline.Runtime_Degraded :=
    VI_Frame.Runtime_Degraded;

VIO_Timeline.Status_Code := VI_Frame.Status_Code;
VIO_Timeline.Status_Text := VI_Frame.Status_Text;

END_FUNCTION_BLOCK
// >>> BULK_SYNC_ANCHOR: FB_Heating_Runtime_Timeline_Observer <<<

(* ---- FB_Heating_Safe_State.st ---- *)
FUNCTION_BLOCK FB_Heating_Safe_State
VAR_INPUT
    VI_Block_Normal_Heating : BOOL;
    VI_IO_Failsafe_Active : BOOL;
    VI_Gas_Safety_Active : BOOL;
    VI_Freeze_Active : BOOL;
    VI_Freeze_Target_Supply : REAL;
    VI_Manifold_Temps_Supply : ARRAY[1..GVL_CONSTANTS.C_MAX_MANIFOLDS] OF REAL;
    VI_Boiler_Error_Status : ARRAY[1..GVL_CONSTANTS.C_MAX_BOILERS] OF BOOL;
    VI_Boiler_OT_Online : ARRAY[1..GVL_CONSTANTS.C_MAX_BOILERS] OF BOOL;
END_VAR
VAR_OUTPUT
    VO_Applied : BOOL;
    VO_Zone_Valves : ARRAY[1..GVL_CONSTANTS.C_MAX_HEATING_CIRCUITS] OF BOOL;
    VO_Manifold_Pumps : ARRAY[1..GVL_CONSTANTS.C_MAX_MANIFOLDS] OF BOOL;
    VO_Manifold_Valves : ARRAY[1..GVL_CONSTANTS.C_MAX_MANIFOLDS] OF REAL;
    VO_Boiler_OT_Enable : ARRAY[1..GVL_CONSTANTS.C_MAX_BOILERS] OF BOOL;
    VO_Boiler_OT_Setpoint : ARRAY[1..GVL_CONSTANTS.C_MAX_BOILERS] OF REAL;
    VO_Boiler_Status : ARRAY[1..GVL_CONSTANTS.C_MAX_BOILERS] OF ST_Boiler_Status;
    VO_Backup_Circulation_Pump : BOOL;
    VO_Electric_Heater_Enable : BOOL;
    VO_Freeze_Risk_Status : BOOL;
END_VAR
VAR
    L_i : INT;
    L_Min_Supply_Temp : REAL;
    L_Freeze_Circulation_Required : BOOL;
END_VAR

VO_Applied := VI_Block_Normal_Heating;
VO_Backup_Circulation_Pump := FALSE;
VO_Electric_Heater_Enable := FALSE;
VO_Freeze_Risk_Status := FALSE;
L_Freeze_Circulation_Required := VI_Freeze_Active AND (VI_IO_Failsafe_Active OR VI_Gas_Safety_Active);

IF NOT VI_Block_Normal_Heating THEN
    RETURN;
END_IF;

FOR L_i := 1 TO GVL_CONSTANTS.C_MAX_HEATING_CIRCUITS DO
    VO_Zone_Valves[L_i] := FALSE;
END_FOR;

FOR L_i := 1 TO GVL_CONSTANTS.C_MAX_MANIFOLDS DO
    IF L_Freeze_Circulation_Required THEN
        VO_Manifold_Pumps[L_i] := TRUE;
        VO_Manifold_Valves[L_i] := REAL#35.0;
    ELSE
        VO_Manifold_Pumps[L_i] := FALSE;
        VO_Manifold_Valves[L_i] := REAL#0.0;
    END_IF;
END_FOR;

FOR L_i := 1 TO GVL_CONSTANTS.C_MAX_BOILERS DO
    VO_Boiler_OT_Enable[L_i] := FALSE;
    VO_Boiler_OT_Setpoint[L_i] := REAL#0.0;
    VO_Boiler_Status[L_i].Warning := FALSE;
    VO_Boiler_Status[L_i].Error := TRUE;
END_FOR;

IF VI_Gas_Safety_Active AND VI_Freeze_Active THEN
    VO_Backup_Circulation_Pump := TRUE;
    L_Min_Supply_Temp := REAL#1000.0;
    FOR L_i := 1 TO GVL_CONSTANTS.C_MAX_MANIFOLDS DO
        IF VI_Manifold_Temps_Supply[L_i] < L_Min_Supply_Temp THEN
            L_Min_Supply_Temp := VI_Manifold_Temps_Supply[L_i];
        END_IF;
    END_FOR;
    IF L_Min_Supply_Temp > REAL#900.0 THEN
        L_Min_Supply_Temp := REAL#0.0;
    END_IF;

    IF L_Min_Supply_Temp < (VI_Freeze_Target_Supply - REAL#1.0) THEN
        VO_Electric_Heater_Enable := TRUE;
    ELSIF L_Min_Supply_Temp > (VI_Freeze_Target_Supply + REAL#1.0) THEN
        VO_Electric_Heater_Enable := FALSE;
    END_IF;
    VO_Freeze_Risk_Status := TRUE;
END_IF;

IF VI_IO_Failsafe_Active AND VI_Freeze_Active THEN
    IF VI_Boiler_OT_Online[1] AND NOT VI_Boiler_Error_Status[1] THEN
        VO_Boiler_OT_Enable[1] := TRUE;
        VO_Boiler_OT_Setpoint[1] := VI_Freeze_Target_Supply;
    END_IF;
END_IF;

END_FUNCTION_BLOCK
// >>> BULK_SYNC_ANCHOR: FB_Heating_Safe_State <<<

(* ---- FB_Heating_Safety_Gate.st ---- *)
// ==============================================================================
// Heating safety gate helper
//
// Internal refactoring helper for FB_Heating_System_Manager.
// Not connected yet. The manager remains the public facade.
// ==============================================================================
FUNCTION_BLOCK FB_Heating_Safety_Gate
VAR_INPUT
    VI_System_Mode : E_System_Operating_Mode;
    VI_Emergency_Stop : BOOL;
    VI_Gas_Safety_Stop : BOOL;
    VI_IO_Failsafe_Active : BOOL;
    VI_Outdoor_Temp : REAL;
    VI_Freeze_Threshold : REAL;
END_VAR

VAR_IN_OUT
    VI_Floor_Temps : ARRAY[1..GVL_CONSTANTS.C_MAX_HEATING_CIRCUITS] OF REAL;
END_VAR

VAR_OUTPUT
    VO_Block_Normal_Heating : BOOL;
    VO_Freeze_Mode_Active : BOOL;
    VO_Freeze_Target_Supply : REAL;
END_VAR

VAR
    L_i : INT;
END_VAR

VO_Block_Normal_Heating := VI_Emergency_Stop OR VI_Gas_Safety_Stop OR VI_IO_Failsafe_Active OR (VI_System_Mode = E_System_Operating_Mode.MODE_SAFE_STOP);
VO_Freeze_Mode_Active := (VI_System_Mode = E_System_Operating_Mode.MODE_FREEZE_PROTECTION) OR (VI_Outdoor_Temp < -5.0);

FOR L_i := 1 TO GVL_CONSTANTS.C_MAX_HEATING_CIRCUITS DO
    IF VI_Floor_Temps[L_i] < 7.0 THEN
        VO_Freeze_Mode_Active := TRUE;
    END_IF;
END_FOR;

IF VO_Freeze_Mode_Active THEN
    VO_Freeze_Target_Supply := LIMIT(20.0, VI_Freeze_Threshold + 2.0, 35.0);
ELSE
    VO_Freeze_Target_Supply := 0.0;
END_IF;

// >>> BULK_SYNC_ANCHOR: FB_Heating_Safety_Gate <<<

(* ---- FB_Heating_Schedule_Preheat.st ---- *)
FUNCTION_BLOCK FB_Heating_Schedule_Preheat
VAR_INPUT
    VI_Time_Of_Day_MS : UDINT;
    VI_Day_Of_Week : INT; // 1=Mon ... 7=Sun
    VI_Enable : BOOL;
END_VAR

VAR
    L_i : INT;
    L_e : INT;
    L_Event : ST_Heating_Schedule_Event;
    L_Time_To_Comfort_MS : UDINT;
    L_Adjustment : REAL;
    L_Max_Boost : REAL;
    L_Active : BOOL;

    L_Learn_Window_MS : UDINT := 300000;
    L_Learn_Cooldown_MS : UDINT := 900000;
    L_Cold_Confirm : ARRAY[1..GVL_CONSTANTS.C_MAX_ZONES, 1..3] OF INT;
    L_Hot_Confirm : ARRAY[1..GVL_CONSTANTS.C_MAX_ZONES, 1..3] OF INT;
    L_Last_Learn_MS : ARRAY[1..GVL_CONSTANTS.C_MAX_ZONES, 1..3] OF UDINT;
END_VAR

IF NOT VI_Enable THEN
    FOR L_i := 1 TO GVL_CONSTANTS.C_MAX_ZONES DO
        GVL_HEATING_POLICY.G_Zone_Schedule_Preheat_Active[L_i] := FALSE;
    END_FOR;
    RETURN;
END_IF;

FOR L_i := 1 TO GVL_CONSTANTS.C_MAX_ZONES DO
    L_Active := FALSE;
    L_Max_Boost := 0.0;

    FOR L_e := 1 TO 3 DO
        L_Event := GVL_HEATING_POLICY_CONFIG.G_Zone_Schedule[L_i, L_e];

        IF L_Event.Enabled THEN
            IF (L_Event.Weekday_Mask AND SHL(1, VI_Day_Of_Week - 1)) <> 0 THEN

                IF L_Event.Comfort_Time_MS >= VI_Time_Of_Day_MS THEN
                    L_Time_To_Comfort_MS := L_Event.Comfort_Time_MS - VI_Time_Of_Day_MS;
                ELSE
                    L_Time_To_Comfort_MS := (86400000 - VI_Time_Of_Day_MS) + L_Event.Comfort_Time_MS;
                END_IF;

                IF L_Event.Adaptive_Enabled THEN
                    IF GVL_HEATING_POLICY.G_Zone_Schedule_Learned_Offset_MS[L_i, L_e] > L_Event.Adaptive_Max_Offset_MS THEN
                        GVL_HEATING_POLICY.G_Zone_Schedule_Learned_Offset_MS[L_i, L_e] := L_Event.Adaptive_Max_Offset_MS;
                    END_IF;
                    L_Time_To_Comfort_MS := L_Time_To_Comfort_MS + GVL_HEATING_POLICY.G_Zone_Schedule_Learned_Offset_MS[L_i, L_e];
                END_IF;

                IF (GVL_HEATING_POLICY.G_Zone_Time_To_Heat_MS[L_i] >= L_Time_To_Comfort_MS)
                   AND (GVL_HEATING_POLICY.G_Zone_Time_To_Heat_MS[L_i] > 0) THEN

                    IF L_Event.Preheat_Boost > L_Max_Boost THEN
                        L_Max_Boost := L_Event.Preheat_Boost;
                    END_IF;

                    L_Active := TRUE;
                END_IF;

                IF L_Event.Adaptive_Enabled THEN
                    IF L_Time_To_Comfort_MS < L_Learn_Window_MS THEN

                        IF GVL_HEATING_POLICY.G_Zone_Thermal_Demand[L_i] > 1.0 THEN
                            L_Cold_Confirm[L_i, L_e] := L_Cold_Confirm[L_i, L_e] + 1;
                            L_Hot_Confirm[L_i, L_e] := 0;
                        ELSIF GVL_HEATING_POLICY.G_Zone_Thermal_Demand[L_i] < -0.5 THEN
                            L_Hot_Confirm[L_i, L_e] := L_Hot_Confirm[L_i, L_e] + 1;
                            L_Cold_Confirm[L_i, L_e] := 0;
                        ELSE
                            L_Cold_Confirm[L_i, L_e] := 0;
                            L_Hot_Confirm[L_i, L_e] := 0;
                        END_IF;

                        IF (VI_Time_Of_Day_MS - L_Last_Learn_MS[L_i, L_e]) >= L_Learn_Cooldown_MS THEN

                            IF L_Cold_Confirm[L_i, L_e] >= 2 THEN
                                IF GVL_HEATING_POLICY.G_Zone_Schedule_Learned_Offset_MS[L_i, L_e] < L_Event.Adaptive_Max_Offset_MS THEN
                                    GVL_HEATING_POLICY.G_Zone_Schedule_Learned_Offset_MS[L_i, L_e] :=
                                        GVL_HEATING_POLICY.G_Zone_Schedule_Learned_Offset_MS[L_i, L_e] + L_Event.Adaptive_Step_MS;
                                    IF GVL_HEATING_POLICY.G_Zone_Schedule_Learned_Offset_MS[L_i, L_e] > L_Event.Adaptive_Max_Offset_MS THEN
                                        GVL_HEATING_POLICY.G_Zone_Schedule_Learned_Offset_MS[L_i, L_e] := L_Event.Adaptive_Max_Offset_MS;
                                    END_IF;
                                    L_Last_Learn_MS[L_i, L_e] := VI_Time_Of_Day_MS;
                                END_IF;
                                L_Cold_Confirm[L_i, L_e] := 0;
                            END_IF;

                            IF L_Hot_Confirm[L_i, L_e] >= 2 THEN
                                IF GVL_HEATING_POLICY.G_Zone_Schedule_Learned_Offset_MS[L_i, L_e] > L_Event.Adaptive_Step_MS THEN
                                    GVL_HEATING_POLICY.G_Zone_Schedule_Learned_Offset_MS[L_i, L_e] :=
                                        GVL_HEATING_POLICY.G_Zone_Schedule_Learned_Offset_MS[L_i, L_e] - L_Event.Adaptive_Step_MS;
                                ELSE
                                    GVL_HEATING_POLICY.G_Zone_Schedule_Learned_Offset_MS[L_i, L_e] := 0;
                                END_IF;
                                L_Last_Learn_MS[L_i, L_e] := VI_Time_Of_Day_MS;
                                L_Hot_Confirm[L_i, L_e] := 0;
                            END_IF;

                        END_IF;
                    ELSE
                        L_Cold_Confirm[L_i, L_e] := 0;
                        L_Hot_Confirm[L_i, L_e] := 0;
                    END_IF;
                END_IF;

            END_IF;
        END_IF;
    END_FOR;

    L_Adjustment := GVL_HEATING_POLICY.G_Zone_Target_Adjustment[L_i];

    IF L_Active AND (L_Adjustment < L_Max_Boost) THEN
        L_Adjustment := L_Max_Boost;
    END_IF;

    IF L_Adjustment > 1.0 THEN
        L_Adjustment := 1.0;
    ELSIF L_Adjustment < -1.0 THEN
        L_Adjustment := -1.0;
    END_IF;

    GVL_HEATING_POLICY.G_Zone_Target_Adjustment[L_i] := L_Adjustment;
    GVL_HEATING_POLICY.G_Zone_Schedule_Preheat_Active[L_i] := L_Active;
END_FOR;

END_FUNCTION_BLOCK
